LIN {X 0,Y 452.591,Z 786.867,A -85,B 0,C 180,E1 7857.223,E2 7857.223} C_VEL
LIN {X 0,Y 442.447,Z 754.81,A -85,B 0,C 180,E1 7858.353,E2 7858.353} C_VEL
LIN {X 0,Y 442.001,Z 754.81,A -85,B 0,C 180,E1 7869.434,E2 7869.434} C_VEL
LIN {X 0,Y 441.88,Z 754.81,A -85,B 0,C 180,E1 7877.96,E2 7877.96} C_VEL
LIN {X 0,Y 441.928,Z 754.81,A -85,B 0,C 180,E1 7887.845,E2 7887.845} C_VEL
LIN {X 0,Y 442.308,Z 754.81,A -85,B 0,C 180,E1 7898.887,E2 7898.887} C_VEL
LIN {X 0,Y 442.704,Z 754.81,A -85,B 0,C 180,E1 7909.135,E2 7909.135} C_VEL
LIN {X 0,Y 443.031,Z 754.81,A -85,B 0,C 180,E1 7919.021,E2 7919.021} C_VEL
LIN {X 0,Y 442.966,Z 754.81,A -85,B 0,C 180,E1 7928.871,E2 7928.871} C_VEL
LIN {X 0,Y 442.439,Z 754.81,A -85,B 0,C 180,E1 7939.392,E2 7939.392} C_VEL
LIN {X 0,Y 442.078,Z 754.81,A -85,B 0,C 180,E1 7949.854,E2 7949.854} C_VEL
LIN {X 0,Y 441.847,Z 754.81,A -85,B 0,C 180,E1 7959.452,E2 7959.452} C_VEL
LIN {X 0,Y 441.828,Z 754.81,A -85,B 0,C 180,E1 7967.949,E2 7967.949} C_VEL
LIN {X 0,Y 441.919,Z 754.81,A -85,B 0,C 180,E1 7977.84,E2 7977.84} C_VEL
LIN {X 0,Y 441.903,Z 754.81,A -85,B 0,C 180,E1 7986.738,E2 7986.738} C_VEL
LIN {X 0,Y 442.395,Z 754.81,A -85,B 0,C 180,E1 7997.116,E2 7997.116} C_VEL
LIN {X 0,Y 443.108,Z 754.81,A -85,B 0,C 180,E1 8007.055,E2 8007.055} C_VEL
LIN {X 0,Y 442.368,Z 756.655,A -85,B 0,C 180,E1 8012.365,E2 8012.365} C_VEL
LIN {X 0,Y 449.575,Z 792.358,A -85,B 0,C 180,E1 8014.536,E2 8014.536} C_VEL
LIN {X 0,Y 447.004,Z 827.238,A -85,B 0,C 180,E1 8018.05,E2 8018.05} C_VEL
LIN {X 0,Y 445.134,Z 851.284,A -85,B 0,C 180,E1 8022.802,E2 8022.802} C_VEL
LIN {X 0,Y 444.477,Z 860.925,A -85,B 0,C 180,E1 8026.87,E2 8026.87} C_VEL
LIN {X 0,Y 444.267,Z 862.934,A -85,B 0,C 180,E1 8031.018,E2 8031.018} C_VEL
LIN {X 0,Y 445.039,Z 852.888,A -85,B 0,C 180,E1 8036.859,E2 8036.859} C_VEL
LIN {X 0,Y 447.157,Z 829.66,A -85,B 0,C 180,E1 8041.738,E2 8041.738} C_VEL
LIN {X 0,Y 449.893,Z 795.07,A -85,B 0,C 180,E1 8045.397,E2 8045.397} C_VEL
LIN {X 0,Y 445.984,Z 767.35,A -85,B 0,C 180,E1 8047.255,E2 8047.255} C_VEL
LIN {X 0,Y 442.165,Z 754.81,A -85,B 0,C 180,E1 8048.173,E2 8048.173} C_VEL
LIN {X 0,Y 441.871,Z 754.81,A -85,B 0,C 180,E1 8057.953,E2 8057.953} C_VEL
LIN {X 0,Y 441.961,Z 754.81,A -85,B 0,C 180,E1 8067.842,E2 8067.842} C_VEL
LIN {X 0,Y 441.936,Z 754.81,A -85,B 0,C 180,E1 8076.738,E2 8076.738} C_VEL
LIN {X 0,Y 442.368,Z 754.81,A -85,B 0,C 180,E1 8087.113,E2 8087.113} C_VEL
LIN {X 0,Y 443.223,Z 754.81,A -85,B 0,C 180,E1 8097.919,E2 8097.919} C_VEL
LIN {X 0,Y 442.747,Z 754.81,A -85,B 0,C 180,E1 8108.87,E2 8108.87} C_VEL
LIN {X 0,Y 442.392,Z 754.81,A -85,B 0,C 180,E1 8119.379,E2 8119.379} C_VEL
LIN {X 0,Y 442.145,Z 754.81,A -85,B 0,C 180,E1 8129.843,E2 8129.843} C_VEL
LIN {X 0,Y 442.036,Z 754.81,A -85,B 0,C 180,E1 8139.426,E2 8139.426} C_VEL
LIN {X 0,Y 441.905,Z 754.81,A -85,B 0,C 180,E1 8147.96,E2 8147.96} C_VEL
LIN {X 0,Y 441.987,Z 754.81,A -85,B 0,C 180,E1 8157.847,E2 8157.847} C_VEL
LIN {X 0,Y 442.617,Z 756.744,A -85,B 0,C 180,E1 8161.684,E2 8161.684} C_VEL
LIN {X 0,Y 454.951,Z 801.269,A -85,B 0,C 180,E1 8163.103,E2 8163.103} C_VEL
LIN {X 0,Y 452.795,Z 857.855,A -85,B 0,C 180,E1 8164.779,E2 8164.779} C_VEL
LIN {X 0,Y 442.938,Z 889.427,A -85,B 0,C 180,E1 8166.427,E2 8166.427} C_VEL
LIN {X 0,Y 438.726,Z 935.255,A -85,B 0,C 180,E1 8171.199,E2 8171.199} C_VEL
LIN {X 0,Y 436.456,Z 968.703,A -85,B 0,C 180,E1 8177.194,E2 8177.194} C_VEL
LIN {X 0,Y 436.059,Z 988.848,A -85,B 0,C 180,E1 8184.008,E2 8184.008} C_VEL
LIN {X 0,Y 435.858,Z 994.128,A -85,B 0,C 180,E1 8190.998,E2 8190.998} C_VEL
LIN {X 0,Y 435.692,Z 985.83,A -85,B 0,C 180,E1 8197.506,E2 8197.506} C_VEL
LIN {X 0,Y 436.647,Z 963.898,A -85,B 0,C 180,E1 8203.956,E2 8203.956} C_VEL
LIN {X 0,Y 439.499,Z 927.872,A -85,B 0,C 180,E1 8209.806,E2 8209.806} C_VEL
LIN {X 0,Y 443.485,Z 882.164,A -85,B 0,C 180,E1 8214.111,E2 8214.111} C_VEL
LIN {X 0,Y 446.96,Z 829.737,A -85,B 0,C 180,E1 8216.636,E2 8216.636} C_VEL
LIN {X 0,Y 445.096,Z 788.288,A -85,B 0,C 180,E1 8217.571,E2 8217.571} C_VEL
LIN {X 0,Y 434.362,Z 754.81,A -85,B 0,C 180,E1 8218.782,E2 8218.782} C_VEL
LIN {X 0,Y 433.933,Z 754.81,A -85,B 0,C 180,E1 8228.11,E2 8228.11} C_VEL
LIN {X 0,Y 433.819,Z 754.81,A -85,B 0,C 180,E1 8238.774,E2 8238.774} C_VEL
LIN {X 0,Y 433.954,Z 754.81,A -85,B 0,C 180,E1 8249.534,E2 8249.534} C_VEL
LIN {X 0,Y 434.39,Z 754.81,A -85,B 0,C 180,E1 8260.62,E2 8260.62} C_VEL
LIN {X 0,Y 434.769,Z 754.81,A -85,B 0,C 180,E1 8270.966,E2 8270.966} C_VEL
LIN {X 0,Y 435.526,Z 754.81,A -85,B 0,C 180,E1 8281.001,E2 8281.001} C_VEL
LIN {X 0,Y 434.752,Z 754.81,A -85,B 0,C 180,E1 8291.071,E2 8291.071} C_VEL
LIN {X 0,Y 434.339,Z 754.81,A -85,B 0,C 180,E1 8301.525,E2 8301.525} C_VEL
LIN {X 0,Y 433.906,Z 754.81,A -85,B 0,C 180,E1 8311.031,E2 8311.031} C_VEL
LIN {X 0,Y 433.754,Z 754.81,A -85,B 0,C 180,E1 8321.216,E2 8321.216} C_VEL
LIN {X 0,Y 433.694,Z 754.81,A -85,B 0,C 180,E1 8331.938,E2 8331.938} C_VEL
LIN {X 0,Y 433.989,Z 754.81,A -85,B 0,C 180,E1 8341.831,E2 8341.831} C_VEL
LIN {X 0,Y 434.256,Z 754.81,A -85,B 0,C 180,E1 8352.719,E2 8352.719} C_VEL
LIN {X 0,Y 434.917,Z 754.81,A -85,B 0,C 180,E1 8362.984,E2 8362.984} C_VEL
LIN {X 0,Y 434.264,Z 754.81,A -85,B 0,C 180,E1 8371.877,E2 8371.877} C_VEL
LIN {X 0,Y 441.972,Z 793.979,A -85,B 0,C 180,E1 8374.278,E2 8374.278} C_VEL
LIN {X 0,Y 439.206,Z 829.188,A -85,B 0,C 180,E1 8377.944,E2 8377.944} C_VEL
LIN {X 0,Y 437.188,Z 853.627,A -85,B 0,C 180,E1 8383.039,E2 8383.039} C_VEL
LIN {X 0,Y 436.52,Z 862.544,A -85,B 0,C 180,E1 8387.187,E2 8387.187} C_VEL
LIN {X 0,Y 436.714,Z 861.813,A -85,B 0,C 180,E1 8393.554,E2 8393.554} C_VEL
LIN {X 0,Y 438.444,Z 845.603,A -85,B 0,C 180,E1 8399.268,E2 8399.268} C_VEL
LIN {X 0,Y 441.034,Z 816.527,A -85,B 0,C 180,E1 8403.848,E2 8403.848} C_VEL
LIN {X 0,Y 441.317,Z 779.381,A -85,B 0,C 180,E1 8406.941,E2 8406.941} C_VEL
LIN {X 0,Y 434.105,Z 754.81,A -85,B 0,C 180,E1 8408.698,E2 8408.698} C_VEL
LIN {X 0,Y 433.757,Z 754.81,A -85,B 0,C 180,E1 8419.663,E2 8419.663} C_VEL
LIN {X 0,Y 433.983,Z 754.81,A -85,B 0,C 180,E1 8429.531,E2 8429.531} C_VEL
LIN {X 0,Y 434.05,Z 754.81,A -85,B 0,C 180,E1 8440.598,E2 8440.598} C_VEL
LIN {X 0,Y 434.799,Z 754.81,A -85,B 0,C 180,E1 8450.961,E2 8450.961} C_VEL
LIN {X 0,Y 435.015,Z 754.81,A -85,B 0,C 180,E1 8460.997,E2 8460.997} C_VEL
LIN {X 0,Y 434.668,Z 754.81,A -85,B 0,C 180,E1 8471.068,E2 8471.068} C_VEL
LIN {X 0,Y 434.322,Z 754.81,A -85,B 0,C 180,E1 8481.52,E2 8481.52} C_VEL
LIN {X 0,Y 433.999,Z 754.81,A -85,B 0,C 180,E1 8491.054,E2 8491.054} C_VEL
LIN {X 0,Y 433.921,Z 754.81,A -85,B 0,C 180,E1 8501.243,E2 8501.243} C_VEL
LIN {X 0,Y 433.89,Z 754.81,A -85,B 0,C 180,E1 8512.261,E2 8512.261} C_VEL
LIN {X 0,Y 434.389,Z 756.03,A -85,B 0,C 180,E1 8521.168,E2 8521.168} C_VEL
LIN {X 0,Y 447.578,Z 800.376,A -85,B 0,C 180,E1 8522.692,E2 8522.692} C_VEL
LIN {X 0,Y 445.33,Z 857.166,A -85,B 0,C 180,E1 8524.398,E2 8524.398} C_VEL
LIN {X 0,Y 442.938,Z 889.427,A -85,B 0,C 180,E1 8526.427,E2 8526.427} C_VEL
LIN {X 0,Y 432.598,Z 917.951,A -85,B 0,C 180,E1 8528.842,E2 8528.842} C_VEL
LIN {X 0,Y 429.325,Z 956.761,A -85,B 0,C 180,E1 8534.627,E2 8534.627} C_VEL
LIN {X 0,Y 427.9,Z 982.008,A -85,B 0,C 180,E1 8541.331,E2 8541.331} C_VEL
LIN {X 0,Y 427.815,Z 991.674,A -85,B 0,C 180,E1 8546.951,E2 8546.951} C_VEL
LIN {X 0,Y 428.118,Z 990.75,A -85,B 0,C 180,E1 8554.066,E2 8554.066} C_VEL
LIN {X 0,Y 428.165,Z 974.434,A -85,B 0,C 180,E1 8561.242,E2 8561.242} C_VEL
LIN {X 0,Y 430.13,Z 944.424,A -85,B 0,C 180,E1 8567.613,E2 8567.613} C_VEL
LIN {X 0,Y 434.112,Z 902.67,A -85,B 0,C 180,E1 8572.723,E2 8572.723} C_VEL
LIN {X 0,Y 438.158,Z 851.791,A -85,B 0,C 180,E1 8576.165,E2 8576.165} C_VEL
LIN {X 0,Y 439.043,Z 794.483,A -85,B 0,C 180,E1 8577.778,E2 8577.778} C_VEL
LIN {X 0,Y 426.256,Z 754.81,A -85,B 0,C 180,E1 8579.285,E2 8579.285} C_VEL
LIN {X 0,Y 425.858,Z 754.81,A -85,B 0,C 180,E1 8589.994,E2 8589.994} C_VEL
LIN {X 0,Y 425.782,Z 754.81,A -85,B 0,C 180,E1 8600.024,E2 8600.024} C_VEL
LIN {X 0,Y 425.936,Z 754.81,A -85,B 0,C 180,E1 8611.253,E2 8611.253} C_VEL
LIN {X 0,Y 426.384,Z 754.81,A -85,B 0,C 180,E1 8622.393,E2 8622.393} C_VEL
LIN {X 0,Y 426.997,Z 754.81,A -85,B 0,C 180,E1 8632.857,E2 8632.857} C_VEL
LIN {X 0,Y 427.048,Z 754.81,A -85,B 0,C 180,E1 8643.058,E2 8643.058} C_VEL
LIN {X 0,Y 426.644,Z 754.81,A -85,B 0,C 180,E1 8653.37,E2 8653.37} C_VEL
LIN {X 0,Y 426.194,Z 754.81,A -85,B 0,C 180,E1 8664.175,E2 8664.175} C_VEL
LIN {X 0,Y 425.794,Z 754.81,A -85,B 0,C 180,E1 8673.537,E2 8673.537} C_VEL
LIN {X 0,Y 425.737,Z 754.81,A -85,B 0,C 180,E1 8684.037,E2 8684.037} C_VEL
LIN {X 0,Y 425.708,Z 754.81,A -85,B 0,C 180,E1 8693.97,E2 8693.97} C_VEL
LIN {X 0,Y 425.968,Z 754.81,A -85,B 0,C 180,E1 8703.555,E2 8703.555} C_VEL
LIN {X 0,Y 426.32,Z 754.81,A -85,B 0,C 180,E1 8714.515,E2 8714.515} C_VEL
LIN {X 0,Y 426.825,Z 754.81,A -85,B 0,C 180,E1 8724.9,E2 8724.9} C_VEL
LIN {X 0,Y 426.509,Z 756.493,A -85,B 0,C 180,E1 8731.529,E2 8731.529} C_VEL
LIN {X 0,Y 434.337,Z 795.975,A -85,B 0,C 180,E1 8734.038,E2 8734.038} C_VEL
LIN {X 0,Y 431.444,Z 831.116,A -85,B 0,C 180,E1 8737.833,E2 8737.833} C_VEL
LIN {X 0,Y 429.385,Z 854.31,A -85,B 0,C 180,E1 8742.761,E2 8742.761} C_VEL
LIN {X 0,Y 428.56,Z 864.155,A -85,B 0,C 180,E1 8747.517,E2 8747.517} C_VEL
LIN {X 0,Y 428.808,Z 863.488,A -85,B 0,C 180,E1 8753.308,E2 8753.308} C_VEL
LIN {X 0,Y 430.356,Z 849.139,A -85,B 0,C 180,E1 8758.923,E2 8758.923} C_VEL
LIN {X 0,Y 433.012,Z 822.26,A -85,B 0,C 180,E1 8763.619,E2 8763.619} C_VEL
LIN {X 0,Y 434.797,Z 785.115,A -85,B 0,C 180,E1 8767.001,E2 8767.001} C_VEL
LIN {X 0,Y 426.077,Z 754.81,A -85,B 0,C 180,E1 8769.059,E2 8769.059} C_VEL
LIN {X 0,Y 425.729,Z 754.81,A -85,B 0,C 180,E1 8780.031,E2 8780.031} C_VEL
LIN {X 0,Y 425.972,Z 754.81,A -85,B 0,C 180,E1 8791.25,E2 8791.25} C_VEL
LIN {X 0,Y 426.174,Z 754.81,A -85,B 0,C 180,E1 8802.379,E2 8802.379} C_VEL
LIN {X 0,Y 426.87,Z 754.81,A -85,B 0,C 180,E1 8812.85,E2 8812.85} C_VEL
LIN {X 0,Y 427.024,Z 754.81,A -85,B 0,C 180,E1 8821.016,E2 8821.016} C_VEL
LIN {X 0,Y 426.647,Z 754.81,A -85,B 0,C 180,E1 8831.279,E2 8831.279} C_VEL
LIN {X 0,Y 426.291,Z 754.81,A -85,B 0,C 180,E1 8841.947,E2 8841.947} C_VEL
LIN {X 0,Y 425.989,Z 754.81,A -85,B 0,C 180,E1 8853.157,E2 8853.157} C_VEL
LIN {X 0,Y 425.864,Z 754.81,A -85,B 0,C 180,E1 8864.014,E2 8864.014} C_VEL
LIN {X 0,Y 425.834,Z 754.81,A -85,B 0,C 180,E1 8873.984,E2 8873.984} C_VEL
LIN {X 0,Y 426.437,Z 756.637,A -85,B 0,C 180,E1 8880.672,E2 8880.672} C_VEL
LIN {X 0,Y 440.238,Z 802.364,A -85,B 0,C 180,E1 8882.317,E2 8882.317} C_VEL
LIN {X 0,Y 437.767,Z 857.949,A -85,B 0,C 180,E1 8884.077,E2 8884.077} C_VEL
LIN {X 0,Y 433.688,Z 907.236,A -85,B 0,C 180,E1 8887.711,E2 8887.711} C_VEL
LIN {X 0,Y 432.598,Z 917.951,A -85,B 0,C 180,E1 8888.842,E2 8888.842} C_VEL
LIN {X 0,Y 422.426,Z 942.481,A -85,B 0,C 180,E1 8891.991,E2 8891.991} C_VEL
LIN {X 0,Y 420.454,Z 973.012,A -85,B 0,C 180,E1 8898.551,E2 8898.551} C_VEL
LIN {X 0,Y 420.028,Z 989.458,A -85,B 0,C 180,E1 8905.857,E2 8905.857} C_VEL
LIN {X 0,Y 420.02,Z 991.768,A -85,B 0,C 180,E1 8911.036,E2 8911.036} C_VEL
LIN {X 0,Y 419.857,Z 983.376,A -85,B 0,C 180,E1 8917.791,E2 8917.791} C_VEL
LIN {X 0,Y 421.142,Z 959.449,A -85,B 0,C 180,E1 8924.878,E2 8924.878} C_VEL
LIN {X 0,Y 424.355,Z 922.522,A -85,B 0,C 180,E1 8930.818,E2 8930.818} C_VEL
LIN {X 0,Y 428.776,Z 874.925,A -85,B 0,C 180,E1 8935.196,E2 8935.196} C_VEL
LIN {X 0,Y 432.221,Z 822.667,A -85,B 0,C 180,E1 8937.566,E2 8937.566} C_VEL
LIN {X 0,Y 430.033,Z 790.74,A -85,B 0,C 180,E1 8938.316,E2 8938.316} C_VEL
LIN {X 0,Y 418.191,Z 754.81,A -85,B 0,C 180,E1 8939.739,E2 8939.739} C_VEL
LIN {X 0,Y 417.841,Z 754.81,A -85,B 0,C 180,E1 8949.465,E2 8949.465} C_VEL
LIN {X 0,Y 417.763,Z 754.81,A -85,B 0,C 180,E1 8960.532,E2 8960.532} C_VEL
LIN {X 0,Y 417.91,Z 754.81,A -85,B 0,C 180,E1 8970.648,E2 8970.648} C_VEL
LIN {X 0,Y 418.354,Z 754.81,A -85,B 0,C 180,E1 8982.044,E2 8982.044} C_VEL
LIN {X 0,Y 418.979,Z 754.81,A -85,B 0,C 180,E1 8992.72,E2 8992.72} C_VEL
LIN {X 0,Y 419.031,Z 754.81,A -85,B 0,C 180,E1 9003.117,E2 9003.117} C_VEL
LIN {X 0,Y 418.611,Z 754.81,A -85,B 0,C 180,E1 9013.632,E2 9013.632} C_VEL
LIN {X 0,Y 418.182,Z 754.81,A -85,B 0,C 180,E1 9024.669,E2 9024.669} C_VEL
LIN {X 0,Y 417.626,Z 754.81,A -85,B 0,C 180,E1 9035.153,E2 9035.153} C_VEL
LIN {X 0,Y 417.7,Z 754.81,A -85,B 0,C 180,E1 9045.113,E2 9045.113} C_VEL
LIN {X 0,Y 417.703,Z 754.81,A -85,B 0,C 180,E1 9055.726,E2 9055.726} C_VEL
LIN {X 0,Y 417.905,Z 754.81,A -85,B 0,C 180,E1 9065.316,E2 9065.316} C_VEL
LIN {X 0,Y 418.308,Z 754.81,A -85,B 0,C 180,E1 9076.36,E2 9076.36} C_VEL
LIN {X 0,Y 419.055,Z 754.81,A -85,B 0,C 180,E1 9086.885,E2 9086.885} C_VEL
LIN {X 0,Y 418.638,Z 756.628,A -85,B 0,C 180,E1 9091.103,E2 9091.103} C_VEL
LIN {X 0,Y 426.819,Z 796.423,A -85,B 0,C 180,E1 9093.676,E2 9093.676} C_VEL
LIN {X 0,Y 423.789,Z 831.313,A -85,B 0,C 180,E1 9097.458,E2 9097.458} C_VEL
LIN {X 0,Y 421.581,Z 854.962,A -85,B 0,C 180,E1 9102.473,E2 9102.473} C_VEL
LIN {X 0,Y 420.616,Z 865.658,A -85,B 0,C 180,E1 9107.858,E2 9107.858} C_VEL
LIN {X 0,Y 421.087,Z 863.073,A -85,B 0,C 180,E1 9114.484,E2 9114.484} C_VEL
LIN {X 0,Y 423.127,Z 846.139,A -85,B 0,C 180,E1 9120.133,E2 9120.133} C_VEL
LIN {X 0,Y 426.134,Z 817.816,A -85,B 0,C 180,E1 9124.615,E2 9124.615} C_VEL
LIN {X 0,Y 426.482,Z 782.61,A -85,B 0,C 180,E1 9127.696,E2 9127.696} C_VEL
LIN {X 0,Y 417.977,Z 754.81,A -85,B 0,C 180,E1 9129.796,E2 9129.796} C_VEL
LIN {X 0,Y 417.703,Z 754.81,A -85,B 0,C 180,E1 9140.518,E2 9140.518} C_VEL
LIN {X 0,Y 417.943,Z 754.81,A -85,B 0,C 180,E1 9150.644,E2 9150.644} C_VEL
LIN {X 0,Y 418.123,Z 754.81,A -85,B 0,C 180,E1 9162.028,E2 9162.028} C_VEL
LIN {X 0,Y 418.851,Z 754.81,A -85,B 0,C 180,E1 9172.712,E2 9172.712} C_VEL
LIN {X 0,Y 419.017,Z 754.81,A -85,B 0,C 180,E1 9181.035,E2 9181.035} C_VEL
LIN {X 0,Y 418.648,Z 754.81,A -85,B 0,C 180,E1 9191.497,E2 9191.497} C_VEL
LIN {X 0,Y 418.226,Z 754.81,A -85,B 0,C 180,E1 9202.393,E2 9202.393} C_VEL
LIN {X 0,Y 417.933,Z 754.81,A -85,B 0,C 180,E1 9211.767,E2 9211.767} C_VEL
LIN {X 0,Y 417.864,Z 754.81,A -85,B 0,C 180,E1 9222.207,E2 9222.207} C_VEL
LIN {X 0,Y 417.835,Z 754.81,A -85,B 0,C 180,E1 9233.183,E2 9233.183} C_VEL
LIN {X 0,Y 418.284,Z 756.272,A -85,B 0,C 180,E1 9240.119,E2 9240.119} C_VEL
LIN {X 0,Y 432.955,Z 804.082,A -85,B 0,C 180,E1 9241.912,E2 9241.912} C_VEL
LIN {X 0,Y 430.197,Z 858.79,A -85,B 0,C 180,E1 9243.743,E2 9243.743} C_VEL
LIN {X 0,Y 425.718,Z 908.98,A -85,B 0,C 180,E1 9247.615,E2 9247.615} C_VEL
LIN {X 0,Y 422.426,Z 942.481,A -85,B 0,C 180,E1 9251.991,E2 9251.991} C_VEL
LIN {X 0,Y 412.724,Z 962.347,A -85,B 0,C 180,E1 9255.822,E2 9255.822} C_VEL
LIN {X 0,Y 412.01,Z 983.167,A -85,B 0,C 180,E1 9262.594,E2 9262.594} C_VEL
LIN {X 0,Y 412.291,Z 990.591,A -85,B 0,C 180,E1 9268.946,E2 9268.946} C_VEL
LIN {X 0,Y 412.076,Z 986.99,A -85,B 0,C 180,E1 9275.283,E2 9275.283} C_VEL
LIN {X 0,Y 412.259,Z 969.907,A -85,B 0,C 180,E1 9282.239,E2 9282.239} C_VEL
LIN {X 0,Y 414.602,Z 938.989,A -85,B 0,C 180,E1 9288.68,E2 9288.68} C_VEL
LIN {X 0,Y 419.144,Z 895.529,A -85,B 0,C 180,E1 9293.896,E2 9293.896} C_VEL
LIN {X 0,Y 423.48,Z 845.445,A -85,B 0,C 180,E1 9297.149,E2 9297.149} C_VEL
LIN {X 0,Y 423.087,Z 794.106,A -85,B 0,C 180,E1 9298.626,E2 9298.626} C_VEL
LIN {X 0,Y 410.116,Z 754.81,A -85,B 0,C 180,E1 9300.236,E2 9300.236} C_VEL
LIN {X 0,Y 409.752,Z 754.81,A -85,B 0,C 180,E1 9310.608,E2 9310.608} C_VEL
LIN {X 0,Y 409.693,Z 754.81,A -85,B 0,C 180,E1 9319.596,E2 9319.596} C_VEL
LIN {X 0,Y 409.889,Z 754.81,A -85,B 0,C 180,E1 9330.468,E2 9330.468} C_VEL
LIN {X 0,Y 410.292,Z 754.81,A -85,B 0,C 180,E1 9341.679,E2 9341.679} C_VEL
LIN {X 0,Y 410.939,Z 754.81,A -85,B 0,C 180,E1 9352.576,E2 9352.576} C_VEL
LIN {X 0,Y 411.028,Z 754.81,A -85,B 0,C 180,E1 9363.177,E2 9363.177} C_VEL
LIN {X 0,Y 410.573,Z 754.81,A -85,B 0,C 180,E1 9373.904,E2 9373.904} C_VEL
LIN {X 0,Y 410.104,Z 754.81,A -85,B 0,C 180,E1 9385.188,E2 9385.188} C_VEL
LIN {X 0,Y 409.635,Z 754.81,A -85,B 0,C 180,E1 9395.048,E2 9395.048} C_VEL
LIN {X 0,Y 409.604,Z 754.81,A -85,B 0,C 180,E1 9406.262,E2 9406.262} C_VEL
LIN {X 0,Y 409.714,Z 754.81,A -85,B 0,C 180,E1 9417.514,E2 9417.514} C_VEL
LIN {X 0,Y 409.823,Z 754.81,A -85,B 0,C 180,E1 9427.118,E2 9427.118} C_VEL
LIN {X 0,Y 410.474,Z 754.81,A -85,B 0,C 180,E1 9438.455,E2 9438.455} C_VEL
LIN {X 0,Y 411.317,Z 754.81,A -85,B 0,C 180,E1 9448.942,E2 9448.942} C_VEL
LIN {X 0,Y 410.806,Z 756.741,A -85,B 0,C 180,E1 9450.661,E2 9450.661} C_VEL
LIN {X 0,Y 419.227,Z 798.212,A -85,B 0,C 180,E1 9453.413,E2 9453.413} C_VEL
LIN {X 0,Y 415.998,Z 833.178,A -85,B 0,C 180,E1 9457.335,E2 9457.335} C_VEL
LIN {X 0,Y 413.678,Z 856.697,A -85,B 0,C 180,E1 9462.529,E2 9462.529} C_VEL
LIN {X 0,Y 412.673,Z 867.156,A -85,B 0,C 180,E1 9468.214,E2 9468.214} C_VEL
LIN {X 0,Y 413.309,Z 863.652,A -85,B 0,C 180,E1 9474.976,E2 9474.976} C_VEL
LIN {X 0,Y 415.625,Z 845.043,A -85,B 0,C 180,E1 9480.897,E2 9480.897} C_VEL
LIN {X 0,Y 419.094,Z 814.777,A -85,B 0,C 180,E1 9485.435,E2 9485.435} C_VEL
LIN {X 0,Y 419.03,Z 784.069,A -85,B 0,C 180,E1 9488.107,E2 9488.107} C_VEL
LIN {X 0,Y 409.923,Z 754.81,A -85,B 0,C 180,E1 9490.38,E2 9490.38} C_VEL
LIN {X 0,Y 409.652,Z 754.81,A -85,B 0,C 180,E1 9499.584,E2 9499.584} C_VEL
LIN {X 0,Y 409.933,Z 754.81,A -85,B 0,C 180,E1 9510.454,E2 9510.454} C_VEL
LIN {X 0,Y 410.046,Z 754.81,A -85,B 0,C 180,E1 9521.662,E2 9521.662} C_VEL
LIN {X 0,Y 410.821,Z 754.81,A -85,B 0,C 180,E1 9532.569,E2 9532.569} C_VEL
LIN {X 0,Y 411.027,Z 754.81,A -85,B 0,C 180,E1 9541.055,E2 9541.055} C_VEL
LIN {X 0,Y 410.63,Z 754.81,A -85,B 0,C 180,E1 9551.725,E2 9551.725} C_VEL
LIN {X 0,Y 410.162,Z 754.81,A -85,B 0,C 180,E1 9562.857,E2 9562.857} C_VEL
LIN {X 0,Y 409.842,Z 754.81,A -85,B 0,C 180,E1 9573.579,E2 9573.579} C_VEL
LIN {X 0,Y 409.716,Z 754.81,A -85,B 0,C 180,E1 9583.758,E2 9583.758} C_VEL
LIN {X 0,Y 409.813,Z 754.81,A -85,B 0,C 180,E1 9594.973,E2 9594.973} C_VEL
LIN {X 0,Y 410.193,Z 756.226,A -85,B 0,C 180,E1 9599.538,E2 9599.538} C_VEL
LIN {X 0,Y 425.692,Z 805.295,A -85,B 0,C 180,E1 9601.484,E2 9601.484} C_VEL
LIN {X 0,Y 422.661,Z 859.766,A -85,B 0,C 180,E1 9603.4,E2 9603.4} C_VEL
LIN {X 0,Y 418.017,Z 908.692,A -85,B 0,C 180,E1 9607.312,E2 9607.312} C_VEL
LIN {X 0,Y 414.12,Z 948.974,A -85,B 0,C 180,E1 9613.013,E2 9613.013} C_VEL
LIN {X 0,Y 412.724,Z 962.347,A -85,B 0,C 180,E1 9615.822,E2 9615.822} C_VEL
LIN {X 0,Y 404.251,Z 976.838,A -85,B 0,C 180,E1 9620.231,E2 9620.231} C_VEL
LIN {X 0,Y 404.086,Z 988.13,A -85,B 0,C 180,E1 9626.771,E2 9626.771} C_VEL
LIN {X 0,Y 404.216,Z 988.182,A -85,B 0,C 180,E1 9633.229,E2 9633.229} C_VEL
LIN {X 0,Y 404.288,Z 973.923,A -85,B 0,C 180,E1 9640.818,E2 9640.818} C_VEL
LIN {X 0,Y 406.174,Z 945.392,A -85,B 0,C 180,E1 9647.696,E2 9647.696} C_VEL
LIN {X 0,Y 410.528,Z 904.705,A -85,B 0,C 180,E1 9653.272,E2 9653.272} C_VEL
LIN {X 0,Y 415.161,Z 855.742,A -85,B 0,C 180,E1 9657.009,E2 9657.009} C_VEL
LIN {X 0,Y 417.289,Z 800.971,A -85,B 0,C 180,E1 9658.822,E2 9658.822} C_VEL
LIN {X 0,Y 402.086,Z 754.81,A -85,B 0,C 180,E1 9660.633,E2 9660.633} C_VEL
LIN {X 0,Y 401.652,Z 754.81,A -85,B 0,C 180,E1 9671.393,E2 9671.393} C_VEL
LIN {X 0,Y 401.636,Z 754.81,A -85,B 0,C 180,E1 9681.436,E2 9681.436} C_VEL
LIN {X 0,Y 401.899,Z 754.81,A -85,B 0,C 180,E1 9692.545,E2 9692.545} C_VEL
LIN {X 0,Y 402.435,Z 754.81,A -85,B 0,C 180,E1 9704.073,E2 9704.073} C_VEL
LIN {X 0,Y 403,Z 754.81,A -85,B 0,C 180,E1 9714.601,E2 9714.601} C_VEL
LIN {X 0,Y 402.965,Z 754.81,A -85,B 0,C 180,E1 9723.618,E2 9723.618} C_VEL
LIN {X 0,Y 402.537,Z 754.81,A -85,B 0,C 180,E1 9734.187,E2 9734.187} C_VEL
LIN {X 0,Y 402.008,Z 754.81,A -85,B 0,C 180,E1 9745.732,E2 9745.732} C_VEL
LIN {X 0,Y 401.594,Z 754.81,A -85,B 0,C 180,E1 9755.857,E2 9755.857} C_VEL
LIN {X 0,Y 401.541,Z 754.81,A -85,B 0,C 180,E1 9765.637,E2 9765.637} C_VEL
LIN {X 0,Y 401.68,Z 754.81,A -85,B 0,C 180,E1 9776.782,E2 9776.782} C_VEL
LIN {X 0,Y 401.776,Z 754.81,A -85,B 0,C 180,E1 9787.734,E2 9787.734} C_VEL
LIN {X 0,Y 402.372,Z 754.81,A -85,B 0,C 180,E1 9798.027,E2 9798.027} C_VEL
LIN {X 0,Y 403.308,Z 754.81,A -85,B 0,C 180,E1 9808.921,E2 9808.921} C_VEL
LIN {X 0,Y 402.997,Z 756.719,A -85,B 0,C 180,E1 9810.202,E2 9810.202} C_VEL
LIN {X 0,Y 411.711,Z 798.72,A -85,B 0,C 180,E1 9813.038,E2 9813.038} C_VEL
LIN {X 0,Y 408.204,Z 834.99,A -85,B 0,C 180,E1 9817.207,E2 9817.207} C_VEL
LIN {X 0,Y 405.732,Z 858.628,A -85,B 0,C 180,E1 9822.671,E2 9822.671} C_VEL
LIN {X 0,Y 404.754,Z 868.556,A -85,B 0,C 180,E1 9828.583,E2 9828.583} C_VEL
LIN {X 0,Y 405.499,Z 864.194,A -85,B 0,C 180,E1 9835.491,E2 9835.491} C_VEL
LIN {X 0,Y 408.027,Z 845.328,A -85,B 0,C 180,E1 9841.364,E2 9841.364} C_VEL
LIN {X 0,Y 411.791,Z 814.569,A -85,B 0,C 180,E1 9845.958,E2 9845.958} C_VEL
LIN {X 0,Y 411.439,Z 784.862,A -85,B 0,C 180,E1 9848.6,E2 9848.6} C_VEL
LIN {X 0,Y 401.862,Z 754.81,A -85,B 0,C 180,E1 9850.93,E2 9850.93} C_VEL
LIN {X 0,Y 401.554,Z 754.81,A -85,B 0,C 180,E1 9861.419,E2 9861.419} C_VEL
LIN {X 0,Y 401.921,Z 754.81,A -85,B 0,C 180,E1 9872.536,E2 9872.536} C_VEL
LIN {X 0,Y 402.205,Z 754.81,A -85,B 0,C 180,E1 9884.183,E2 9884.183} C_VEL
LIN {X 0,Y 402.777,Z 754.81,A -85,B 0,C 180,E1 9894.592,E2 9894.592} C_VEL
LIN {X 0,Y 402.859,Z 754.81,A -85,B 0,C 180,E1 9903.395,E2 9903.395} C_VEL
LIN {X 0,Y 402.511,Z 754.81,A -85,B 0,C 180,E1 9914.183,E2 9914.183} C_VEL
LIN {X 0,Y 402.019,Z 754.81,A -85,B 0,C 180,E1 9925.725,E2 9925.725} C_VEL
LIN {X 0,Y 401.854,Z 754.81,A -85,B 0,C 180,E1 9935.823,E2 9935.823} C_VEL
LIN {X 0,Y 401.625,Z 754.81,A -85,B 0,C 180,E1 9947.456,E2 9947.456} C_VEL
LIN {X 0,Y 402.141,Z 756.322,A -85,B 0,C 180,E1 9958.936,E2 9958.936} C_VEL
LIN {X 0,Y 418.44,Z 806.325,A -85,B 0,C 180,E1 9961.041,E2 9961.041} C_VEL
LIN {X 0,Y 415.096,Z 860.998,A -85,B 0,C 180,E1 9963.069,E2 9963.069} C_VEL
LIN {X 0,Y 410.139,Z 909.749,A -85,B 0,C 180,E1 9967.139,E2 9967.139} C_VEL
LIN {X 0,Y 406.149,Z 949.193,A -85,B 0,C 180,E1 9972.97,E2 9972.97} C_VEL
LIN {X 0,Y 404.251,Z 976.838,A -85,B 0,C 180,E1 9980.231,E2 9980.231} C_VEL
LIN {X 0,Y 396.308,Z 985.239,A -85,B 0,C 180,E1 9985.053,E2 9985.053} C_VEL
LIN {X 0,Y 396.278,Z 988.222,A -85,B 0,C 180,E1 9991.098,E2 9991.098} C_VEL
LIN {X 0,Y 396.126,Z 979.622,A -85,B 0,C 180,E1 9998.261,E2 9998.261} C_VEL
LIN {X 0,Y 397.634,Z 955.186,A -85,B 0,C 180,E1 10005.78,E2 10005.78} C_VEL
LIN {X 0,Y 401.316,Z 917.733,A -85,B 0,C 180,E1 10012.012,E2 10012.012} C_VEL
LIN {X 0,Y 406.253,Z 870.749,A -85,B 0,C 180,E1 10016.451,E2 10016.451} C_VEL
LIN {X 0,Y 409.994,Z 816.866,A -85,B 0,C 180,E1 10018.891,E2 10018.891} C_VEL
LIN {X 0,Y 406.9,Z 792.819,A -85,B 0,C 180,E1 10019.557,E2 10019.557} C_VEL
LIN {X 0,Y 393.957,Z 754.81,A -85,B 0,C 180,E1 10021.336,E2 10021.336} C_VEL
LIN {X 0,Y 393.636,Z 754.81,A -85,B 0,C 180,E1 10032.43,E2 10032.43} C_VEL
LIN {X 0,Y 393.566,Z 754.81,A -85,B 0,C 180,E1 10043.301,E2 10043.301} C_VEL
LIN {X 0,Y 393.861,Z 754.81,A -85,B 0,C 180,E1 10053.702,E2 10053.702} C_VEL
LIN {X 0,Y 394.524,Z 754.81,A -85,B 0,C 180,E1 10065.524,E2 10065.524} C_VEL
LIN {X 0,Y 394.929,Z 754.81,A -85,B 0,C 180,E1 10076.699,E2 10076.699} C_VEL
LIN {X 0,Y 394.807,Z 754.81,A -85,B 0,C 180,E1 10085.517,E2 10085.517} C_VEL
LIN {X 0,Y 394.46,Z 754.81,A -85,B 0,C 180,E1 10096.773,E2 10096.773} C_VEL
LIN {X 0,Y 393.972,Z 754.81,A -85,B 0,C 180,E1 10106.297,E2 10106.297} C_VEL
LIN {X 0,Y 393.442,Z 754.81,A -85,B 0,C 180,E1 10117.746,E2 10117.746} C_VEL
LIN {X 0,Y 393.498,Z 754.81,A -85,B 0,C 180,E1 10128.771,E2 10128.771} C_VEL
LIN {X 0,Y 393.68,Z 754.81,A -85,B 0,C 180,E1 10140.155,E2 10140.155} C_VEL
LIN {X 0,Y 393.917,Z 754.81,A -85,B 0,C 180,E1 10150.884,E2 10150.884} C_VEL
LIN {X 0,Y 394.784,Z 754.81,A -85,B 0,C 180,E1 10162.267,E2 10162.267} C_VEL
LIN {X 0,Y 395.137,Z 756.551,A -85,B 0,C 180,E1 10169.724,E2 10169.724} C_VEL
LIN {X 0,Y 404.219,Z 799.197,A -85,B 0,C 180,E1 10172.647,E2 10172.647} C_VEL
LIN {X 0,Y 400.612,Z 835.152,A -85,B 0,C 180,E1 10176.798,E2 10176.798} C_VEL
LIN {X 0,Y 398.035,Z 858.532,A -85,B 0,C 180,E1 10182.104,E2 10182.104} C_VEL
LIN {X 0,Y 397.113,Z 867.986,A -85,B 0,C 180,E1 10186.655,E2 10186.655} C_VEL
LIN {X 0,Y 396.892,Z 870.065,A -85,B 0,C 180,E1 10191.299,E2 10191.299} C_VEL
LIN {X 0,Y 398.267,Z 860.374,A -85,B 0,C 180,E1 10197.852,E2 10197.852} C_VEL
LIN {X 0,Y 401.542,Z 837.06,A -85,B 0,C 180,E1 10203.477,E2 10203.477} C_VEL
LIN {X 0,Y 405.641,Z 802.15,A -85,B 0,C 180,E1 10207.684,E2 10207.684} C_VEL
LIN {X 0,Y 398.278,Z 767.296,A -85,B 0,C 180,E1 10210.541,E2 10210.541} C_VEL
LIN {X 0,Y 393.746,Z 754.81,A -85,B 0,C 180,E1 10211.506,E2 10211.506} C_VEL
LIN {X 0,Y 393.482,Z 754.81,A -85,B 0,C 180,E1 10222.244,E2 10222.244} C_VEL
LIN {X 0,Y 393.859,Z 754.81,A -85,B 0,C 180,E1 10233.695,E2 10233.695} C_VEL
LIN {X 0,Y 394.201,Z 754.81,A -85,B 0,C 180,E1 10245.506,E2 10245.506} C_VEL
LIN {X 0,Y 395.033,Z 754.81,A -85,B 0,C 180,E1 10256.694,E2 10256.694} C_VEL
LIN {X 0,Y 394.801,Z 754.81,A -85,B 0,C 180,E1 10267.729,E2 10267.729} C_VEL
LIN {X 0,Y 394.22,Z 754.81,A -85,B 0,C 180,E1 10279.096,E2 10279.096} C_VEL
LIN {X 0,Y 393.802,Z 754.81,A -85,B 0,C 180,E1 10289.881,E2 10289.881} C_VEL
LIN {X 0,Y 393.666,Z 754.81,A -85,B 0,C 180,E1 10301.261,E2 10301.261} C_VEL
LIN {X 0,Y 393.597,Z 754.81,A -85,B 0,C 180,E1 10312.218,E2 10312.218} C_VEL
LIN {X 0,Y 394.046,Z 756.395,A -85,B 0,C 180,E1 10318.295,E2 10318.295} C_VEL
LIN {X 0,Y 411.265,Z 806.215,A -85,B 0,C 180,E1 10320.551,E2 10320.551} C_VEL
LIN {X 0,Y 407.812,Z 859.868,A -85,B 0,C 180,E1 10322.582,E2 10322.582} C_VEL
LIN {X 0,Y 402.614,Z 908.427,A -85,B 0,C 180,E1 10326.686,E2 10326.686} C_VEL
LIN {X 0,Y 398.242,Z 948.306,A -85,B 0,C 180,E1 10332.694,E2 10332.694} C_VEL
LIN {X 0,Y 396.34,Z 975.755,A -85,B 0,C 180,E1 10340.079,E2 10340.079} C_VEL
LIN {X 0,Y 396.308,Z 985.239,A -85,B 0,C 180,E1 10345.053,E2 10345.053} C_VEL
LIN {X 0,Y 388.356,Z 987.04,A -85,B 0,C 180,E1 10350.099,E2 10350.099} C_VEL
LIN {X 0,Y 388.098,Z 980.553,A -85,B 0,C 180,E1 10357.302,E2 10357.302} C_VEL
LIN {X 0,Y 389.043,Z 959.667,A -85,B 0,C 180,E1 10364.689,E2 10364.689} C_VEL
LIN {X 0,Y 392.661,Z 923.893,A -85,B 0,C 180,E1 10371.393,E2 10371.393} C_VEL
LIN {X 0,Y 397.956,Z 877.456,A -85,B 0,C 180,E1 10376.306,E2 10376.306} C_VEL
LIN {X 0,Y 402.276,Z 824.719,A -85,B 0,C 180,E1 10379.086,E2 10379.086} C_VEL
LIN {X 0,Y 400.131,Z 796.385,A -85,B 0,C 180,E1 10379.888,E2 10379.888} C_VEL
LIN {X 0,Y 385.873,Z 754.81,A -85,B 0,C 180,E1 10381.741,E2 10381.741} C_VEL
LIN {X 0,Y 385.601,Z 754.81,A -85,B 0,C 180,E1 10393.531,E2 10393.531} C_VEL
LIN {X 0,Y 385.554,Z 754.81,A -85,B 0,C 180,E1 10405.203,E2 10405.203} C_VEL
LIN {X 0,Y 385.886,Z 754.81,A -85,B 0,C 180,E1 10415.614,E2 10415.614} C_VEL
LIN {X 0,Y 386.46,Z 754.81,A -85,B 0,C 180,E1 10425.215,E2 10425.215} C_VEL
LIN {X 0,Y 386.942,Z 754.81,A -85,B 0,C 180,E1 10436.63,E2 10436.63} C_VEL
LIN {X 0,Y 386.795,Z 754.81,A -85,B 0,C 180,E1 10445.632,E2 10445.632} C_VEL
LIN {X 0,Y 386.398,Z 754.81,A -85,B 0,C 180,E1 10457.134,E2 10457.134} C_VEL
LIN {X 0,Y 385.804,Z 754.81,A -85,B 0,C 180,E1 10467.741,E2 10467.741} C_VEL
LIN {X 0,Y 385.472,Z 754.81,A -85,B 0,C 180,E1 10479.851,E2 10479.851} C_VEL
LIN {X 0,Y 385.468,Z 754.81,A -85,B 0,C 180,E1 10490.152,E2 10490.152} C_VEL
LIN {X 0,Y 385.687,Z 754.81,A -85,B 0,C 180,E1 10500.537,E2 10500.537} C_VEL
LIN {X 0,Y 385.872,Z 754.81,A -85,B 0,C 180,E1 10510.47,E2 10510.47} C_VEL
LIN {X 0,Y 386.748,Z 754.81,A -85,B 0,C 180,E1 10522.105,E2 10522.105} C_VEL
LIN {X 0,Y 387.267,Z 756.214,A -85,B 0,C 180,E1 10529.22,E2 10529.22} C_VEL
LIN {X 0,Y 396.769,Z 799.189,A -85,B 0,C 180,E1 10532.21,E2 10532.21} C_VEL
LIN {X 0,Y 393.017,Z 835.232,A -85,B 0,C 180,E1 10536.373,E2 10536.373} C_VEL
LIN {X 0,Y 390.234,Z 859.126,A -85,B 0,C 180,E1 10541.78,E2 10541.78} C_VEL
LIN {X 0,Y 389.123,Z 869.764,A -85,B 0,C 180,E1 10547.151,E2 10547.151} C_VEL
LIN {X 0,Y 389.49,Z 869.104,A -85,B 0,C 180,E1 10554.148,E2 10554.148} C_VEL
LIN {X 0,Y 392.046,Z 853.63,A -85,B 0,C 180,E1 10560.534,E2 10560.534} C_VEL
LIN {X 0,Y 396.054,Z 825.206,A -85,B 0,C 180,E1 10565.769,E2 10565.769} C_VEL
LIN {X 0,Y 397.257,Z 790.368,A -85,B 0,C 180,E1 10569.293,E2 10569.293} C_VEL
LIN {X 0,Y 385.686,Z 754.81,A -85,B 0,C 180,E1 10572.207,E2 10572.207} C_VEL
LIN {X 0,Y 385.475,Z 754.81,A -85,B 0,C 180,E1 10583.809,E2 10583.809} C_VEL
LIN {X 0,Y 385.77,Z 754.81,A -85,B 0,C 180,E1 10593.1,E2 10593.1} C_VEL
LIN {X 0,Y 386.149,Z 754.81,A -85,B 0,C 180,E1 10605.197,E2 10605.197} C_VEL
LIN {X 0,Y 387.03,Z 754.81,A -85,B 0,C 180,E1 10616.625,E2 10616.625} C_VEL
LIN {X 0,Y 386.765,Z 754.81,A -85,B 0,C 180,E1 10627.89,E2 10627.89} C_VEL
LIN {X 0,Y 386.195,Z 754.81,A -85,B 0,C 180,E1 10639.509,E2 10639.509} C_VEL
LIN {X 0,Y 385.839,Z 754.81,A -85,B 0,C 180,E1 10649.445,E2 10649.445} C_VEL
LIN {X 0,Y 385.661,Z 754.81,A -85,B 0,C 180,E1 10660.482,E2 10660.482} C_VEL
LIN {X 0,Y 385.576,Z 754.81,A -85,B 0,C 180,E1 10670.124,E2 10670.124} C_VEL
LIN {X 0,Y 385.996,Z 756.415,A -85,B 0,C 180,E1 10677.614,E2 10677.614} C_VEL
LIN {X 0,Y 404.087,Z 806.071,A -85,B 0,C 180,E1 10680.037,E2 10680.037} C_VEL
LIN {X 0,Y 400.468,Z 859.833,A -85,B 0,C 180,E1 10682.133,E2 10682.133} C_VEL
LIN {X 0,Y 394.9,Z 908.366,A -85,B 0,C 180,E1 10686.363,E2 10686.363} C_VEL
LIN {X 0,Y 390.412,Z 946.56,A -85,B 0,C 180,E1 10692.227,E2 10692.227} C_VEL
LIN {X 0,Y 388.515,Z 973.124,A -85,B 0,C 180,E1 10699.308,E2 10699.308} C_VEL
LIN {X 0,Y 388.266,Z 985.781,A -85,B 0,C 180,E1 10706.64,E2 10706.64} C_VEL
LIN {X 0,Y 388.356,Z 987.04,A -85,B 0,C 180,E1 10710.099,E2 10710.099} C_VEL
LIN {X 0,Y 380.358,Z 982.676,A -85,B 0,C 180,E1 10715.242,E2 10715.242} C_VEL
LIN {X 0,Y 380.412,Z 966.392,A -85,B 0,C 180,E1 10722.675,E2 10722.675} C_VEL
LIN {X 0,Y 383.104,Z 935.915,A -85,B 0,C 180,E1 10729.677,E2 10729.677} C_VEL
LIN {X 0,Y 388.501,Z 892.927,A -85,B 0,C 180,E1 10735.294,E2 10735.294} C_VEL
LIN {X 0,Y 393.66,Z 842.438,A -85,B 0,C 180,E1 10738.809,E2 10738.809} C_VEL
LIN {X 0,Y 393.442,Z 800.442,A -85,B 0,C 180,E1 10740.21,E2 10740.21} C_VEL
LIN {X 0,Y 377.84,Z 754.81,A -85,B 0,C 180,E1 10742.101,E2 10742.101} C_VEL
LIN {X 0,Y 377.503,Z 754.81,A -85,B 0,C 180,E1 10751.958,E2 10751.958} C_VEL
LIN {X 0,Y 377.507,Z 754.81,A -85,B 0,C 180,E1 10761.62,E2 10761.62} C_VEL
LIN {X 0,Y 377.735,Z 754.81,A -85,B 0,C 180,E1 10772.486,E2 10772.486} C_VEL
LIN {X 0,Y 378.219,Z 754.81,A -85,B 0,C 180,E1 10782.49,E2 10782.49} C_VEL
LIN {X 0,Y 378.947,Z 754.81,A -85,B 0,C 180,E1 10794.257,E2 10794.257} C_VEL
LIN {X 0,Y 379.019,Z 754.81,A -85,B 0,C 180,E1 10803.446,E2 10803.446} C_VEL
LIN {X 0,Y 378.467,Z 754.81,A -85,B 0,C 180,E1 10815.111,E2 10815.111} C_VEL
LIN {X 0,Y 377.864,Z 754.81,A -85,B 0,C 180,E1 10825.357,E2 10825.357} C_VEL
LIN {X 0,Y 377.41,Z 754.81,A -85,B 0,C 180,E1 10835.668,E2 10835.668} C_VEL
LIN {X 0,Y 377.375,Z 754.81,A -85,B 0,C 180,E1 10845.271,E2 10845.271} C_VEL
LIN {X 0,Y 377.521,Z 754.81,A -85,B 0,C 180,E1 10857.133,E2 10857.133} C_VEL
LIN {X 0,Y 377.703,Z 754.81,A -85,B 0,C 180,E1 10867.56,E2 10867.56} C_VEL
LIN {X 0,Y 378.518,Z 754.81,A -85,B 0,C 180,E1 10879.605,E2 10879.605} C_VEL
LIN {X 0,Y 379.349,Z 755.935,A -85,B 0,C 180,E1 10888.695,E2 10888.695} C_VEL
LIN {X 0,Y 389.26,Z 799.657,A -85,B 0,C 180,E1 10891.797,E2 10891.797} C_VEL
LIN {X 0,Y 385.447,Z 835.256,A -85,B 0,C 180,E1 10895.931,E2 10895.931} C_VEL
LIN {X 0,Y 382.451,Z 859.681,A -85,B 0,C 180,E1 10901.443,E2 10901.443} C_VEL
LIN {X 0,Y 381.189,Z 871.185,A -85,B 0,C 180,E1 10907.372,E2 10907.372} C_VEL
LIN {X 0,Y 381.402,Z 871.511,A -85,B 0,C 180,E1 10913.117,E2 10913.117} C_VEL
LIN {X 0,Y 383.569,Z 858.941,A -85,B 0,C 180,E1 10919.64,E2 10919.64} C_VEL
LIN {X 0,Y 387.593,Z 832.997,A -85,B 0,C 180,E1 10925.238,E2 10925.238} C_VEL
LIN {X 0,Y 390.696,Z 795.565,A -85,B 0,C 180,E1 10929.423,E2 10929.423} C_VEL
LIN {X 0,Y 377.603,Z 754.81,A -85,B 0,C 180,E1 10932.937,E2 10932.937} C_VEL
LIN {X 0,Y 377.469,Z 754.81,A -85,B 0,C 180,E1 10944.338,E2 10944.338} C_VEL
LIN {X 0,Y 377.732,Z 754.81,A -85,B 0,C 180,E1 10955.046,E2 10955.046} C_VEL
LIN {X 0,Y 378.132,Z 754.81,A -85,B 0,C 180,E1 10964.876,E2 10964.876} C_VEL
LIN {X 0,Y 379.007,Z 754.81,A -85,B 0,C 180,E1 10976.554,E2 10976.554} C_VEL
LIN {X 0,Y 378.731,Z 754.81,A -85,B 0,C 180,E1 10988.059,E2 10988.059} C_VEL
LIN {X 0,Y 378.127,Z 754.81,A -85,B 0,C 180,E1 10999.943,E2 10999.943} C_VEL
LIN {X 0,Y 377.724,Z 754.81,A -85,B 0,C 180,E1 11010.255,E2 11010.255} C_VEL
LIN {X 0,Y 377.524,Z 754.81,A -85,B 0,C 180,E1 11021.957,E2 11021.957} C_VEL
LIN {X 0,Y 377.545,Z 754.81,A -85,B 0,C 180,E1 11031.606,E2 11031.606} C_VEL
LIN {X 0,Y 377.989,Z 756.612,A -85,B 0,C 180,E1 11036.906,E2 11036.906} C_VEL
LIN {X 0,Y 396.963,Z 809.107,A -85,B 0,C 180,E1 11039.578,E2 11039.578} C_VEL
LIN {X 0,Y 392.829,Z 862.483,A -85,B 0,C 180,E1 11041.834,E2 11041.834} C_VEL
LIN {X 0,Y 386.985,Z 910.338,A -85,B 0,C 180,E1 11046.26,E2 11046.26} C_VEL
LIN {X 0,Y 382.257,Z 949.289,A -85,B 0,C 180,E1 11052.678,E2 11052.678} C_VEL
LIN {X 0,Y 380.389,Z 974.821,A -85,B 0,C 180,E1 11060.239,E2 11060.239} C_VEL
LIN {X 0,Y 380.34,Z 984.608,A -85,B 0,C 180,E1 11066.569,E2 11066.569} C_VEL
LIN {X 0,Y 380.474,Z 984.571,A -85,B 0,C 180,E1 11073.431,E2 11073.431} C_VEL
LIN {X 0,Y 380.358,Z 982.676,A -85,B 0,C 180,E1 11075.242,E2 11075.242} C_VEL
LIN {X 0,Y 372.466,Z 972.403,A -85,B 0,C 180,E1 11080.292,E2 11080.292} C_VEL
LIN {X 0,Y 374.173,Z 946.606,A -85,B 0,C 180,E1 11087.71,E2 11087.71} C_VEL
LIN {X 0,Y 379.106,Z 906.86,A -85,B 0,C 180,E1 11094.068,E2 11094.068} C_VEL
LIN {X 0,Y 384.642,Z 858.602,A -85,B 0,C 180,E1 11098.34,E2 11098.34} C_VEL
LIN {X 0,Y 387.176,Z 805.895,A -85,B 0,C 180,E1 11100.483,E2 11100.483} C_VEL
LIN {X 0,Y 369.747,Z 754.81,A -85,B 0,C 180,E1 11102.719,E2 11102.719} C_VEL
LIN {X 0,Y 369.394,Z 754.81,A -85,B 0,C 180,E1 11114.038,E2 11114.038} C_VEL
LIN {X 0,Y 369.413,Z 754.81,A -85,B 0,C 180,E1 11123.444,E2 11123.444} C_VEL
LIN {X 0,Y 369.745,Z 754.81,A -85,B 0,C 180,E1 11134.475,E2 11134.475} C_VEL
LIN {X 0,Y 370.353,Z 754.81,A -85,B 0,C 180,E1 11144.556,E2 11144.556} C_VEL
LIN {X 0,Y 370.951,Z 754.81,A -85,B 0,C 180,E1 11156.485,E2 11156.485} C_VEL
LIN {X 0,Y 370.773,Z 754.81,A -85,B 0,C 180,E1 11165.876,E2 11165.876} C_VEL
LIN {X 0,Y 370.377,Z 754.81,A -85,B 0,C 180,E1 11175.657,E2 11175.657} C_VEL
LIN {X 0,Y 369.853,Z 754.81,A -85,B 0,C 180,E1 11185.523,E2 11185.523} C_VEL
LIN {X 0,Y 369.312,Z 754.81,A -85,B 0,C 180,E1 11196.745,E2 11196.745} C_VEL
LIN {X 0,Y 369.291,Z 754.81,A -85,B 0,C 180,E1 11207.307,E2 11207.307} C_VEL
LIN {X 0,Y 369.508,Z 754.81,A -85,B 0,C 180,E1 11219.11,E2 11219.11} C_VEL
LIN {X 0,Y 369.729,Z 754.81,A -85,B 0,C 180,E1 11229.58,E2 11229.58} C_VEL
LIN {X 0,Y 370.676,Z 754.81,A -85,B 0,C 180,E1 11241.761,E2 11241.761} C_VEL
LIN {X 0,Y 371.384,Z 756.601,A -85,B 0,C 180,E1 11248.184,E2 11248.184} C_VEL
LIN {X 0,Y 381.379,Z 799.501,A -85,B 0,C 180,E1 11251.287,E2 11251.287} C_VEL
LIN {X 0,Y 377.927,Z 835.263,A -85,B 0,C 180,E1 11255.472,E2 11255.472} C_VEL
LIN {X 0,Y 374.687,Z 860.231,A -85,B 0,C 180,E1 11261.091,E2 11261.091} C_VEL
LIN {X 0,Y 373.233,Z 872.679,A -85,B 0,C 180,E1 11267.754,E2 11267.754} C_VEL
LIN {X 0,Y 373.972,Z 870.523,A -85,B 0,C 180,E1 11275.219,E2 11275.219} C_VEL
LIN {X 0,Y 377.06,Z 853.608,A -85,B 0,C 180,E1 11281.782,E2 11281.782} C_VEL
LIN {X 0,Y 381.745,Z 824.389,A -85,B 0,C 180,E1 11287.031,E2 11287.031} C_VEL
LIN {X 0,Y 382.753,Z 794.101,A -85,B 0,C 180,E1 11290.224,E2 11290.224} C_VEL
LIN {X 0,Y 369.55,Z 754.81,A -85,B 0,C 180,E1 11293.763,E2 11293.763} C_VEL
LIN {X 0,Y 369.372,Z 754.81,A -85,B 0,C 180,E1 11303.432,E2 11303.432} C_VEL
LIN {X 0,Y 369.704,Z 754.81,A -85,B 0,C 180,E1 11314.466,E2 11314.466} C_VEL
LIN {X 0,Y 370.072,Z 754.81,A -85,B 0,C 180,E1 11324.538,E2 11324.538} C_VEL
LIN {X 0,Y 371,Z 754.81,A -85,B 0,C 180,E1 11336.479,E2 11336.479} C_VEL
LIN {X 0,Y 370.882,Z 754.81,A -85,B 0,C 180,E1 11345.868,E2 11345.868} C_VEL
LIN {X 0,Y 370.189,Z 754.81,A -85,B 0,C 180,E1 11357.903,E2 11357.903} C_VEL
LIN {X 0,Y 369.748,Z 754.81,A -85,B 0,C 180,E1 11368.16,E2 11368.16} C_VEL
LIN {X 0,Y 369.489,Z 754.81,A -85,B 0,C 180,E1 11379.536,E2 11379.536} C_VEL
LIN {X 0,Y 369.399,Z 754.81,A -85,B 0,C 180,E1 11390.449,E2 11390.449} C_VEL
LIN {X 0,Y 369.883,Z 756.545,A -85,B 0,C 180,E1 11396.134,E2 11396.134} C_VEL
LIN {X 0,Y 389.741,Z 808.975,A -85,B 0,C 180,E1 11399.011,E2 11399.011} C_VEL
LIN {X 0,Y 385.538,Z 862.147,A -85,B 0,C 180,E1 11401.333,E2 11401.333} C_VEL
LIN {X 0,Y 379.416,Z 909.441,A -85,B 0,C 180,E1 11405.797,E2 11405.797} C_VEL
LIN {X 0,Y 374.376,Z 948.091,A -85,B 0,C 180,E1 11412.302,E2 11412.302} C_VEL
LIN {X 0,Y 372.443,Z 973.651,A -85,B 0,C 180,E1 11420.028,E2 11420.028} C_VEL
LIN {X 0,Y 372.425,Z 983.55,A -85,B 0,C 180,E1 11426.628,E2 11426.628} C_VEL
LIN {X 0,Y 372.546,Z 983.22,A -85,B 0,C 180,E1 11433.675,E2 11433.675} C_VEL
LIN {X 0,Y 372.466,Z 972.403,A -85,B 0,C 180,E1 11440.292,E2 11440.292} C_VEL
LIN {X 0,Y 365.294,Z 957.214,A -85,B 0,C 180,E1 11445.151,E2 11445.151} C_VEL
LIN {X 0,Y 369.201,Z 922.783,A -85,B 0,C 180,E1 11452.143,E2 11452.143} C_VEL
LIN {X 0,Y 374.965,Z 878.069,A -85,B 0,C 180,E1 11457.298,E2 11457.298} C_VEL
LIN {X 0,Y 379.883,Z 826.258,A -85,B 0,C 180,E1 11460.321,E2 11460.321} C_VEL
LIN {X 0,Y 378.026,Z 801.847,A -85,B 0,C 180,E1 11461.155,E2 11461.155} C_VEL
LIN {X 0,Y 361.697,Z 754.81,A -85,B 0,C 180,E1 11463.464,E2 11463.464} C_VEL
LIN {X 0,Y 361.388,Z 754.81,A -85,B 0,C 180,E1 11473.86,E2 11473.86} C_VEL
LIN {X 0,Y 361.387,Z 754.81,A -85,B 0,C 180,E1 11485.47,E2 11485.47} C_VEL
LIN {X 0,Y 361.805,Z 754.81,A -85,B 0,C 180,E1 11496.521,E2 11496.521} C_VEL
LIN {X 0,Y 362.429,Z 754.81,A -85,B 0,C 180,E1 11506.689,E2 11506.689} C_VEL
LIN {X 0,Y 362.939,Z 754.81,A -85,B 0,C 180,E1 11516.407,E2 11516.407} C_VEL
LIN {X 0,Y 362.757,Z 754.81,A -85,B 0,C 180,E1 11526.006,E2 11526.006} C_VEL
LIN {X 0,Y 362.37,Z 754.81,A -85,B 0,C 180,E1 11535.799,E2 11535.799} C_VEL
LIN {X 0,Y 361.766,Z 754.81,A -85,B 0,C 180,E1 11546.136,E2 11546.136} C_VEL
LIN {X 0,Y 361.225,Z 754.81,A -85,B 0,C 180,E1 11557.533,E2 11557.533} C_VEL
LIN {X 0,Y 361.268,Z 754.81,A -85,B 0,C 180,E1 11569.374,E2 11569.374} C_VEL
LIN {X 0,Y 361.488,Z 754.81,A -85,B 0,C 180,E1 11581.132,E2 11581.132} C_VEL
LIN {X 0,Y 361.835,Z 754.81,A -85,B 0,C 180,E1 11591.665,E2 11591.665} C_VEL
LIN {X 0,Y 362.636,Z 754.81,A -85,B 0,C 180,E1 11601.577,E2 11601.577} C_VEL
LIN {X 0,Y 363.221,Z 756.142,A -85,B 0,C 180,E1 11607.605,E2 11607.605} C_VEL
LIN {X 0,Y 373.506,Z 799.563,A -85,B 0,C 180,E1 11610.776,E2 11610.776} C_VEL
LIN {X 0,Y 370.425,Z 835.271,A -85,B 0,C 180,E1 11614.994,E2 11614.994} C_VEL
LIN {X 0,Y 366.951,Z 860.774,A -85,B 0,C 180,E1 11620.725,E2 11620.725} C_VEL
LIN {X 0,Y 365.476,Z 872.668,A -85,B 0,C 180,E1 11626.513,E2 11626.513} C_VEL
LIN {X 0,Y 365.618,Z 874.013,A -85,B 0,C 180,E1 11633.223,E2 11633.223} C_VEL
LIN {X 0,Y 368.227,Z 861.349,A -85,B 0,C 180,E1 11640.211,E2 11640.211} C_VEL
LIN {X 0,Y 372.928,Z 834.848,A -85,B 0,C 180,E1 11646.16,E2 11646.16} C_VEL
LIN {X 0,Y 376.031,Z 798.281,A -85,B 0,C 180,E1 11650.468,E2 11650.468} C_VEL
LIN {X 0,Y 362.06,Z 757.834,A -85,B 0,C 180,E1 11654.217,E2 11654.217} C_VEL
LIN {X 0,Y 361.395,Z 754.81,A -85,B 0,C 180,E1 11654.743,E2 11654.743} C_VEL
LIN {X 0,Y 361.36,Z 754.81,A -85,B 0,C 180,E1 11665.459,E2 11665.459} C_VEL
LIN {X 0,Y 361.644,Z 754.81,A -85,B 0,C 180,E1 11676.503,E2 11676.503} C_VEL
LIN {X 0,Y 362.13,Z 754.81,A -85,B 0,C 180,E1 11686.671,E2 11686.671} C_VEL
LIN {X 0,Y 363.437,Z 754.81,A -85,B 0,C 180,E1 11698.801,E2 11698.801} C_VEL
LIN {X 0,Y 362.527,Z 754.81,A -85,B 0,C 180,E1 11710.855,E2 11710.855} C_VEL
LIN {X 0,Y 362.02,Z 754.81,A -85,B 0,C 180,E1 11720.871,E2 11720.871} C_VEL
LIN {X 0,Y 361.626,Z 754.81,A -85,B 0,C 180,E1 11731.635,E2 11731.635} C_VEL
LIN {X 0,Y 361.411,Z 754.81,A -85,B 0,C 180,E1 11743.85,E2 11743.85} C_VEL
LIN {X 0,Y 361.705,Z 756.001,A -85,B 0,C 180,E1 11755.294,E2 11755.294} C_VEL
LIN {X 0,Y 382.872,Z 811.625,A -85,B 0,C 180,E1 11758.518,E2 11758.518} C_VEL
LIN {X 0,Y 377.952,Z 864.97,A -85,B 0,C 180,E1 11761.032,E2 11761.032} C_VEL
LIN {X 0,Y 371.25,Z 912.673,A -85,B 0,C 180,E1 11765.873,E2 11765.873} C_VEL
LIN {X 0,Y 366.306,Z 949.644,A -85,B 0,C 180,E1 11772.556,E2 11772.556} C_VEL
LIN {X 0,Y 364.439,Z 973.738,A -85,B 0,C 180,E1 11780.413,E2 11780.413} C_VEL
LIN {X 0,Y 364.506,Z 982.277,A -85,B 0,C 180,E1 11786.42,E2 11786.42} C_VEL
LIN {X 0,Y 364.631,Z 982.137,A -85,B 0,C 180,E1 11793.58,E2 11793.58} C_VEL
LIN {X 0,Y 364.42,Z 968.994,A -85,B 0,C 180,E1 11801.349,E2 11801.349} C_VEL
LIN {X 0,Y 365.294,Z 957.214,A -85,B 0,C 180,E1 11805.151,E2 11805.151} C_VEL
LIN {X 0,Y 359.119,Z 937.531,A -85,B 0,C 180,E1 11809.731,E2 11809.731} C_VEL
LIN {X 0,Y 364.861,Z 896.133,A -85,B 0,C 180,E1 11815.896,E2 11815.896} C_VEL
LIN {X 0,Y 370.836,Z 846.695,A -85,B 0,C 180,E1 11819.863,E2 11819.863} C_VEL
LIN {X 0,Y 371.344,Z 805.612,A -85,B 0,C 180,E1 11821.503,E2 11821.503} C_VEL
LIN {X 0,Y 353.614,Z 754.81,A -85,B 0,C 180,E1 11823.991,E2 11823.991} C_VEL
LIN {X 0,Y 353.313,Z 754.81,A -85,B 0,C 180,E1 11835.132,E2 11835.132} C_VEL
LIN {X 0,Y 353.344,Z 754.81,A -85,B 0,C 180,E1 11846.879,E2 11846.879} C_VEL
LIN {X 0,Y 353.867,Z 754.81,A -85,B 0,C 180,E1 11858.625,E2 11858.625} C_VEL
LIN {X 0,Y 354.507,Z 754.81,A -85,B 0,C 180,E1 11868.897,E2 11868.897} C_VEL
LIN {X 0,Y 355.451,Z 754.81,A -85,B 0,C 180,E1 11881.226,E2 11881.226} C_VEL
LIN {X 0,Y 354.413,Z 754.81,A -85,B 0,C 180,E1 11893.624,E2 11893.624} C_VEL
LIN {X 0,Y 353.849,Z 754.81,A -85,B 0,C 180,E1 11904.047,E2 11904.047} C_VEL
LIN {X 0,Y 353.237,Z 754.81,A -85,B 0,C 180,E1 11915.453,E2 11915.453} C_VEL
LIN {X 0,Y 353.224,Z 754.81,A -85,B 0,C 180,E1 11925.149,E2 11925.149} C_VEL
LIN {X 0,Y 353.336,Z 754.81,A -85,B 0,C 180,E1 11937.528,E2 11937.528} C_VEL
LIN {X 0,Y 353.617,Z 754.81,A -85,B 0,C 180,E1 11948.605,E2 11948.605} C_VEL
LIN {X 0,Y 354.372,Z 754.81,A -85,B 0,C 180,E1 11958.888,E2 11958.888} C_VEL
LIN {X 0,Y 355.245,Z 756.474,A -85,B 0,C 180,E1 11967.032,E2 11967.032} C_VEL
LIN {X 0,Y 365.719,Z 799.976,A -85,B 0,C 180,E1 11970.293,E2 11970.293} C_VEL
LIN {X 0,Y 362.663,Z 837.018,A -85,B 0,C 180,E1 11974.8,E2 11974.8} C_VEL
LIN {X 0,Y 358.933,Z 863.107,A -85,B 0,C 180,E1 11980.967,E2 11980.967} C_VEL
LIN {X 0,Y 357.474,Z 874.6,A -85,B 0,C 180,E1 11987.211,E2 11987.211} C_VEL
LIN {X 0,Y 357.998,Z 874.409,A -85,B 0,C 180,E1 11994.295,E2 11994.295} C_VEL
LIN {X 0,Y 361.162,Z 860.216,A -85,B 0,C 180,E1 12001.274,E2 12001.274} C_VEL
LIN {X 0,Y 366.226,Z 832.587,A -85,B 0,C 180,E1 12007.148,E2 12007.148} C_VEL
LIN {X 0,Y 368.545,Z 798.951,A -85,B 0,C 180,E1 12011.109,E2 12011.109} C_VEL
LIN {X 0,Y 354.649,Z 759.124,A -85,B 0,C 180,E1 12014.968,E2 12014.968} C_VEL
LIN {X 0,Y 353.347,Z 754.81,A -85,B 0,C 180,E1 12015.649,E2 12015.649} C_VEL
LIN {X 0,Y 353.362,Z 754.81,A -85,B 0,C 180,E1 12027.529,E2 12027.529} C_VEL
LIN {X 0,Y 353.645,Z 754.81,A -85,B 0,C 180,E1 12038.605,E2 12038.605} C_VEL
LIN {X 0,Y 354.346,Z 754.81,A -85,B 0,C 180,E1 12048.885,E2 12048.885} C_VEL
LIN {X 0,Y 355.443,Z 754.81,A -85,B 0,C 180,E1 12058.774,E2 12058.774} C_VEL
LIN {X 0,Y 354.483,Z 754.81,A -85,B 0,C 180,E1 12071.104,E2 12071.104} C_VEL
LIN {X 0,Y 353.886,Z 754.81,A -85,B 0,C 180,E1 12082.784,E2 12082.784} C_VEL
LIN {X 0,Y 353.464,Z 754.81,A -85,B 0,C 180,E1 12093.154,E2 12093.154} C_VEL
LIN {X 0,Y 353.33,Z 754.81,A -85,B 0,C 180,E1 12105.123,E2 12105.123} C_VEL
LIN {X 0,Y 353.718,Z 756.594,A -85,B 0,C 180,E1 12114.453,E2 12114.453} C_VEL
LIN {X 0,Y 375.536,Z 811.624,A -85,B 0,C 180,E1 12117.893,E2 12117.893} C_VEL
LIN {X 0,Y 370.818,Z 863.786,A -85,B 0,C 180,E1 12120.419,E2 12120.419} C_VEL
LIN {X 0,Y 363.969,Z 910.452,A -85,B 0,C 180,E1 12125.194,E2 12125.194} C_VEL
LIN {X 0,Y 358.507,Z 947.794,A -85,B 0,C 180,E1 12131.989,E2 12131.989} C_VEL
LIN {X 0,Y 356.504,Z 972.593,A -85,B 0,C 180,E1 12140.197,E2 12140.197} C_VEL
LIN {X 0,Y 356.739,Z 982.237,A -85,B 0,C 180,E1 12148.425,E2 12148.425} C_VEL
LIN {X 0,Y 356.463,Z 978.28,A -85,B 0,C 180,E1 12156.111,E2 12156.111} C_VEL
LIN {X 0,Y 356.872,Z 960.253,A -85,B 0,C 180,E1 12164.154,E2 12164.154} C_VEL
LIN {X 0,Y 359.119,Z 937.531,A -85,B 0,C 180,E1 12169.731,E2 12169.731} C_VEL
LIN {X 0,Y 354.72,Z 913.86,A -85,B 0,C 180,E1 12173.93,E2 12173.93} C_VEL
LIN {X 0,Y 360.951,Z 867.6,A -85,B 0,C 180,E1 12178.915,E2 12178.915} C_VEL
LIN {X 0,Y 365.682,Z 814.46,A -85,B 0,C 180,E1 12181.637,E2 12181.637} C_VEL
LIN {X 0,Y 345.527,Z 754.81,A -85,B 0,C 180,E1 12184.613,E2 12184.613} C_VEL
LIN {X 0,Y 345.2,Z 754.81,A -85,B 0,C 180,E1 12197.051,E2 12197.051} C_VEL
LIN {X 0,Y 345.334,Z 754.81,A -85,B 0,C 180,E1 12208.975,E2 12208.975} C_VEL
LIN {X 0,Y 345.956,Z 754.81,A -85,B 0,C 180,E1 12220.796,E2 12220.796} C_VEL
LIN {X 0,Y 346.667,Z 754.81,A -85,B 0,C 180,E1 12231.19,E2 12231.19} C_VEL
LIN {X 0,Y 347.432,Z 754.81,A -85,B 0,C 180,E1 12241.255,E2 12241.255} C_VEL
LIN {X 0,Y 346.388,Z 754.81,A -85,B 0,C 180,E1 12253.946,E2 12253.946} C_VEL
LIN {X 0,Y 345.625,Z 754.81,A -85,B 0,C 180,E1 12265.825,E2 12265.825} C_VEL
LIN {X 0,Y 345.184,Z 754.81,A -85,B 0,C 180,E1 12276.41,E2 12276.41} C_VEL
LIN {X 0,Y 345.115,Z 754.81,A -85,B 0,C 180,E1 12287.032,E2 12287.032} C_VEL
LIN {X 0,Y 345.292,Z 754.81,A -85,B 0,C 180,E1 12298.99,E2 12298.99} C_VEL
LIN {X 0,Y 345.697,Z 754.81,A -85,B 0,C 180,E1 12310.776,E2 12310.776} C_VEL
LIN {X 0,Y 346.556,Z 754.81,A -85,B 0,C 180,E1 12321.183,E2 12321.183} C_VEL
LIN {X 0,Y 347.189,Z 756.563,A -85,B 0,C 180,E1 12326.426,E2 12326.426} C_VEL
LIN {X 0,Y 357.514,Z 798.03,A -85,B 0,C 180,E1 12329.555,E2 12329.555} C_VEL
LIN {X 0,Y 356.613,Z 827.959,A -85,B 0,C 180,E1 12332.931,E2 12332.931} C_VEL
LIN {X 0,Y 352.394,Z 857.388,A -85,B 0,C 180,E1 12338.668,E2 12338.668} C_VEL
LIN {X 0,Y 349.914,Z 873.257,A -85,B 0,C 180,E1 12345.082,E2 12345.082} C_VEL
LIN {X 0,Y 349.538,Z 877.269,A -85,B 0,C 180,E1 12351.656,E2 12351.656} C_VEL
LIN {X 0,Y 351.712,Z 868.191,A -85,B 0,C 180,E1 12359.143,E2 12359.143} C_VEL
LIN {X 0,Y 356.666,Z 844.809,A -85,B 0,C 180,E1 12365.732,E2 12365.732} C_VEL
LIN {X 0,Y 362.628,Z 809.492,A -85,B 0,C 180,E1 12370.637,E2 12370.637} C_VEL
LIN {X 0,Y 352.141,Z 771.035,A -85,B 0,C 180,E1 12374.758,E2 12374.758} C_VEL
LIN {X 0,Y 345.312,Z 754.81,A -85,B 0,C 180,E1 12376.479,E2 12376.479} C_VEL
LIN {X 0,Y 345.337,Z 754.81,A -85,B 0,C 180,E1 12388.971,E2 12388.971} C_VEL
LIN {X 0,Y 345.712,Z 754.81,A -85,B 0,C 180,E1 12400.775,E2 12400.775} C_VEL
LIN {X 0,Y 346.525,Z 754.81,A -85,B 0,C 180,E1 12411.18,E2 12411.18} C_VEL
LIN {X 0,Y 347.022,Z 754.81,A -85,B 0,C 180,E1 12421.25,E2 12421.25} C_VEL
LIN {X 0,Y 346.459,Z 754.81,A -85,B 0,C 180,E1 12431.365,E2 12431.365} C_VEL
LIN {X 0,Y 345.899,Z 754.81,A -85,B 0,C 180,E1 12441.892,E2 12441.892} C_VEL
LIN {X 0,Y 345.446,Z 754.81,A -85,B 0,C 180,E1 12453.303,E2 12453.303} C_VEL
LIN {X 0,Y 345.24,Z 754.81,A -85,B 0,C 180,E1 12463.508,E2 12463.508} C_VEL
LIN {X 0,Y 345.534,Z 756.302,A -85,B 0,C 180,E1 12473.5,E2 12473.5} C_VEL
LIN {X 0,Y 368.212,Z 811.831,A -85,B 0,C 180,E1 12477.243,E2 12477.243} C_VEL
LIN {X 0,Y 363.491,Z 864.556,A -85,B 0,C 180,E1 12479.935,E2 12479.935} C_VEL
LIN {X 0,Y 356.155,Z 911.541,A -85,B 0,C 180,E1 12484.949,E2 12484.949} C_VEL
LIN {X 0,Y 350.452,Z 948.637,A -85,B 0,C 180,E1 12492.07,E2 12492.07} C_VEL
LIN {X 0,Y 348.502,Z 972.702,A -85,B 0,C 180,E1 12500.603,E2 12500.603} C_VEL
LIN {X 0,Y 348.902,Z 981.138,A -85,B 0,C 180,E1 12508.755,E2 12508.755} C_VEL
LIN {X 0,Y 348.524,Z 977.002,A -85,B 0,C 180,E1 12516.25,E2 12516.25} C_VEL
LIN {X 0,Y 349.028,Z 958.781,A -85,B 0,C 180,E1 12524.479,E2 12524.479} C_VEL
LIN {X 0,Y 352.938,Z 925.715,A -85,B 0,C 180,E1 12532.058,E2 12532.058} C_VEL
LIN {X 0,Y 354.72,Z 913.86,A -85,B 0,C 180,E1 12533.93,E2 12533.93} C_VEL
LIN {X 0,Y 350.816,Z 886.707,A -85,B 0,C 180,E1 12537.586,E2 12537.586} C_VEL
LIN {X 0,Y 356.971,Z 835.89,A -85,B 0,C 180,E1 12541.316,E2 12541.316} C_VEL
LIN {X 0,Y 356.177,Z 807.458,A -85,B 0,C 180,E1 12542.498,E2 12542.498} C_VEL
LIN {X 0,Y 337.455,Z 754.81,A -85,B 0,C 180,E1 12545.289,E2 12545.289} C_VEL
LIN {X 0,Y 337.11,Z 754.81,A -85,B 0,C 180,E1 12557.97,E2 12557.97} C_VEL
LIN {X 0,Y 337.324,Z 754.81,A -85,B 0,C 180,E1 12568.849,E2 12568.849} C_VEL
LIN {X 0,Y 337.901,Z 754.81,A -85,B 0,C 180,E1 12580.319,E2 12580.319} C_VEL
LIN {X 0,Y 338.639,Z 754.81,A -85,B 0,C 180,E1 12590.979,E2 12590.979} C_VEL
LIN {X 0,Y 339.418,Z 754.81,A -85,B 0,C 180,E1 12601.284,E2 12601.284} C_VEL
LIN {X 0,Y 338.5,Z 754.81,A -85,B 0,C 180,E1 12611.642,E2 12611.642} C_VEL
LIN {X 0,Y 337.777,Z 754.81,A -85,B 0,C 180,E1 12622.921,E2 12622.921} C_VEL
LIN {X 0,Y 337.193,Z 754.81,A -85,B 0,C 180,E1 12634.237,E2 12634.237} C_VEL
LIN {X 0,Y 337.033,Z 754.81,A -85,B 0,C 180,E1 12645.738,E2 12645.738} C_VEL
LIN {X 0,Y 337.258,Z 754.81,A -85,B 0,C 180,E1 12656.356,E2 12656.356} C_VEL
LIN {X 0,Y 337.502,Z 754.81,A -85,B 0,C 180,E1 12667.529,E2 12667.529} C_VEL
LIN {X 0,Y 338.262,Z 754.81,A -85,B 0,C 180,E1 12678.352,E2 12678.352} C_VEL
LIN {X 0,Y 339.054,Z 756.606,A -85,B 0,C 180,E1 12685.788,E2 12685.788} C_VEL
LIN {X 0,Y 349.609,Z 797.55,A -85,B 0,C 180,E1 12688.933,E2 12688.933} C_VEL
LIN {X 0,Y 349.871,Z 822.952,A -85,B 0,C 180,E1 12691.744,E2 12691.744} C_VEL
LIN {X 0,Y 345.153,Z 854.89,A -85,B 0,C 180,E1 12697.469,E2 12697.469} C_VEL
LIN {X 0,Y 342.242,Z 873.001,A -85,B 0,C 180,E1 12704.115,E2 12704.115} C_VEL
LIN {X 0,Y 341.735,Z 878.33,A -85,B 0,C 180,E1 12712.176,E2 12712.176} C_VEL
LIN {X 0,Y 344.193,Z 868.728,A -85,B 0,C 180,E1 12719.736,E2 12719.736} C_VEL
LIN {X 0,Y 349.568,Z 844.964,A -85,B 0,C 180,E1 12726.409,E2 12726.409} C_VEL
LIN {X 0,Y 355.364,Z 808.883,A -85,B 0,C 180,E1 12731.446,E2 12731.446} C_VEL
LIN {X 0,Y 343.417,Z 769.01,A -85,B 0,C 180,E1 12735.886,E2 12735.886} C_VEL
LIN {X 0,Y 337.178,Z 754.81,A -85,B 0,C 180,E1 12737.497,E2 12737.497} C_VEL
LIN {X 0,Y 337.326,Z 754.81,A -85,B 0,C 180,E1 12748.841,E2 12748.841} C_VEL
LIN {X 0,Y 337.662,Z 754.81,A -85,B 0,C 180,E1 12760.298,E2 12760.298} C_VEL
LIN {X 0,Y 338.503,Z 754.81,A -85,B 0,C 180,E1 12770.969,E2 12770.969} C_VEL
LIN {X 0,Y 339.028,Z 754.81,A -85,B 0,C 180,E1 12781.279,E2 12781.279} C_VEL
LIN {X 0,Y 338.409,Z 754.81,A -85,B 0,C 180,E1 12791.639,E2 12791.639} C_VEL
LIN {X 0,Y 337.763,Z 754.81,A -85,B 0,C 180,E1 12802.919,E2 12802.919} C_VEL
LIN {X 0,Y 337.379,Z 754.81,A -85,B 0,C 180,E1 12814.208,E2 12814.208} C_VEL
LIN {X 0,Y 337.15,Z 754.81,A -85,B 0,C 180,E1 12825.76,E2 12825.76} C_VEL
LIN {X 0,Y 337.449,Z 755.987,A -85,B 0,C 180,E1 12832.498,E2 12832.498} C_VEL
LIN {X 0,Y 360.819,Z 811.671,A -85,B 0,C 180,E1 12836.529,E2 12836.529} C_VEL
LIN {X 0,Y 356.497,Z 863.468,A -85,B 0,C 180,E1 12839.282,E2 12839.282} C_VEL
LIN {X 0,Y 348.76,Z 910.461,A -85,B 0,C 180,E1 12844.38,E2 12844.38} C_VEL
LIN {X 0,Y 342.62,Z 947.323,A -85,B 0,C 180,E1 12851.589,E2 12851.589} C_VEL
LIN {X 0,Y 340.545,Z 971.561,A -85,B 0,C 180,E1 12860.381,E2 12860.381} C_VEL
LIN {X 0,Y 340.99,Z 979.958,A -85,B 0,C 180,E1 12868.726,E2 12868.726} C_VEL
LIN {X 0,Y 340.589,Z 975.723,A -85,B 0,C 180,E1 12876.396,E2 12876.396} C_VEL
LIN {X 0,Y 341.172,Z 957.305,A -85,B 0,C 180,E1 12884.82,E2 12884.82} C_VEL
LIN {X 0,Y 345.287,Z 924.361,A -85,B 0,C 180,E1 12892.482,E2 12892.482} C_VEL
LIN {X 0,Y 350.816,Z 886.707,A -85,B 0,C 180,E1 12897.586,E2 12897.586} C_VEL
LIN {X 0,Y 347.288,Z 856.51,A -85,B 0,C 180,E1 12900.591,E2 12900.591} C_VEL
LIN {X 0,Y 349.41,Z 811.075,A -85,B 0,C 180,E1 12902.883,E2 12902.883} C_VEL
LIN {X 0,Y 329.457,Z 754.81,A -85,B 0,C 180,E1 12905.862,E2 12905.862} C_VEL
LIN {X 0,Y 329.107,Z 754.81,A -85,B 0,C 180,E1 12918.045,E2 12918.045} C_VEL
LIN {X 0,Y 329.312,Z 754.81,A -85,B 0,C 180,E1 12928.491,E2 12928.491} C_VEL
LIN {X 0,Y 329.889,Z 754.81,A -85,B 0,C 180,E1 12940.573,E2 12940.573} C_VEL
LIN {X 0,Y 330.798,Z 754.81,A -85,B 0,C 180,E1 12953.418,E2 12953.418} C_VEL
LIN {X 0,Y 330.91,Z 754.81,A -85,B 0,C 180,E1 12963.948,E2 12963.948} C_VEL
LIN {X 0,Y 330.306,Z 754.81,A -85,B 0,C 180,E1 12974.64,E2 12974.64} C_VEL
LIN {X 0,Y 329.547,Z 754.81,A -85,B 0,C 180,E1 12986.104,E2 12986.104} C_VEL
LIN {X 0,Y 328.999,Z 754.81,A -85,B 0,C 180,E1 12998.518,E2 12998.518} C_VEL
LIN {X 0,Y 328.993,Z 754.81,A -85,B 0,C 180,E1 13009.566,E2 13009.566} C_VEL
LIN {X 0,Y 329.299,Z 754.81,A -85,B 0,C 180,E1 13021.059,E2 13021.059} C_VEL
LIN {X 0,Y 329.75,Z 754.81,A -85,B 0,C 180,E1 13032.593,E2 13032.593} C_VEL
LIN {X 0,Y 330.803,Z 755.339,A -85,B 0,C 180,E1 13045.065,E2 13045.065} C_VEL
LIN {X 0,Y 341.636,Z 796.048,A -85,B 0,C 180,E1 13048.201,E2 13048.201} C_VEL
LIN {X 0,Y 342.539,Z 822.156,A -85,B 0,C 180,E1 13051.11,E2 13051.11} C_VEL
LIN {X 0,Y 337.563,Z 854.525,A -85,B 0,C 180,E1 13056.822,E2 13056.822} C_VEL
LIN {X 0,Y 334.491,Z 873.298,A -85,B 0,C 180,E1 13063.539,E2 13063.539} C_VEL
LIN {X 0,Y 333.71,Z 879.722,A -85,B 0,C 180,E1 13071.204,E2 13071.204} C_VEL
LIN {X 0,Y 335.948,Z 872.092,A -85,B 0,C 180,E1 13079.051,E2 13079.051} C_VEL
LIN {X 0,Y 341.356,Z 849.998,A -85,B 0,C 180,E1 13086.108,E2 13086.108} C_VEL
LIN {X 0,Y 348.162,Z 815.187,A -85,B 0,C 180,E1 13091.469,E2 13091.469} C_VEL
LIN {X 0,Y 339.612,Z 778.614,A -85,B 0,C 180,E1 13095.824,E2 13095.824} C_VEL
LIN {X 0,Y 329.101,Z 754.81,A -85,B 0,C 180,E1 13098.442,E2 13098.442} C_VEL
LIN {X 0,Y 329.355,Z 754.81,A -85,B 0,C 180,E1 13111.062,E2 13111.062} C_VEL
LIN {X 0,Y 329.746,Z 754.81,A -85,B 0,C 180,E1 13122.59,E2 13122.59} C_VEL
LIN {X 0,Y 330.598,Z 754.81,A -85,B 0,C 180,E1 13133.407,E2 13133.407} C_VEL
LIN {X 0,Y 331.019,Z 754.81,A -85,B 0,C 180,E1 13141.31,E2 13141.31} C_VEL
LIN {X 0,Y 330.363,Z 754.81,A -85,B 0,C 180,E1 13151.926,E2 13151.926} C_VEL
LIN {X 0,Y 329.761,Z 754.81,A -85,B 0,C 180,E1 13163.023,E2 13163.023} C_VEL
LIN {X 0,Y 329.236,Z 754.81,A -85,B 0,C 180,E1 13175.177,E2 13175.177} C_VEL
LIN {X 0,Y 329.141,Z 754.81,A -85,B 0,C 180,E1 13185.61,E2 13185.61} C_VEL
LIN {X 0,Y 329.514,Z 756.715,A -85,B 0,C 180,E1 13191.474,E2 13191.474} C_VEL
LIN {X 0,Y 353.349,Z 811.201,A -85,B 0,C 180,E1 13195.76,E2 13195.76} C_VEL
LIN {X 0,Y 351.751,Z 848.47,A -85,B 0,C 180,E1 13197.64,E2 13197.64} C_VEL
LIN {X 0,Y 343.75,Z 896.886,A -85,B 0,C 180,E1 13202.057,E2 13202.057} C_VEL
LIN {X 0,Y 336.087,Z 936.878,A -85,B 0,C 180,E1 13208.825,E2 13208.825} C_VEL
LIN {X 0,Y 332.711,Z 963.45,A -85,B 0,C 180,E1 13216.818,E2 13216.818} C_VEL
LIN {X 0,Y 332.771,Z 976.619,A -85,B 0,C 180,E1 13224.768,E2 13224.768} C_VEL
LIN {X 0,Y 332.99,Z 978.647,A -85,B 0,C 180,E1 13231.307,E2 13231.307} C_VEL
LIN {X 0,Y 332.722,Z 970.384,A -85,B 0,C 180,E1 13239.187,E2 13239.187} C_VEL
LIN {X 0,Y 334.265,Z 946.109,A -85,B 0,C 180,E1 13247.977,E2 13247.977} C_VEL
LIN {X 0,Y 339.921,Z 908.263,A -85,B 0,C 180,E1 13255.273,E2 13255.273} C_VEL
LIN {X 0,Y 346.617,Z 861.585,A -85,B 0,C 180,E1 13260.233,E2 13260.233} C_VEL
LIN {X 0,Y 347.288,Z 856.51,A -85,B 0,C 180,E1 13260.591,E2 13260.591} C_VEL
LIN {X 0,Y 343.174,Z 823.944,A -85,B 0,C 180,E1 13262.841,E2 13262.841} C_VEL
LIN {X 0,Y 331.169,Z 781.086,A -85,B 0,C 180,E1 13265.022,E2 13265.022} C_VEL
LIN {X 0,Y 321.314,Z 754.81,A -85,B 0,C 180,E1 13266.691,E2 13266.691} C_VEL
LIN {X 0,Y 321.057,Z 754.81,A -85,B 0,C 180,E1 13277.111,E2 13277.111} C_VEL
LIN {X 0,Y 321.131,Z 754.81,A -85,B 0,C 180,E1 13287.085,E2 13287.085} C_VEL
LIN {X 0,Y 321.723,Z 754.81,A -85,B 0,C 180,E1 13299.286,E2 13299.286} C_VEL
LIN {X 0,Y 322.586,Z 754.81,A -85,B 0,C 180,E1 13310.527,E2 13310.527} C_VEL
LIN {X 0,Y 323.385,Z 754.81,A -85,B 0,C 180,E1 13321.348,E2 13321.348} C_VEL
LIN {X 0,Y 322.391,Z 754.81,A -85,B 0,C 180,E1 13332.233,E2 13332.233} C_VEL
LIN {X 0,Y 321.653,Z 754.81,A -85,B 0,C 180,E1 13343.646,E2 13343.646} C_VEL
LIN {X 0,Y 321.013,Z 754.81,A -85,B 0,C 180,E1 13356.227,E2 13356.227} C_VEL
LIN {X 0,Y 320.962,Z 754.81,A -85,B 0,C 180,E1 13367.132,E2 13367.132} C_VEL
LIN {X 0,Y 321.073,Z 754.81,A -85,B 0,C 180,E1 13377.073,E2 13377.073} C_VEL
LIN {X 0,Y 321.5,Z 754.81,A -85,B 0,C 180,E1 13389.266,E2 13389.266} C_VEL
LIN {X 0,Y 322.439,Z 754.81,A -85,B 0,C 180,E1 13400.518,E2 13400.518} C_VEL
LIN {X 0,Y 322.798,Z 756.164,A -85,B 0,C 180,E1 13404.392,E2 13404.392} C_VEL
LIN {X 0,Y 333.895,Z 795.957,A -85,B 0,C 180,E1 13407.585,E2 13407.585} C_VEL
LIN {X 0,Y 335.084,Z 822.745,A -85,B 0,C 180,E1 13410.637,E2 13410.637} C_VEL
LIN {X 0,Y 329.923,Z 854.514,A -85,B 0,C 180,E1 13416.271,E2 13416.271} C_VEL
LIN {X 0,Y 326.667,Z 874.003,A -85,B 0,C 180,E1 13423.19,E2 13423.19} C_VEL
LIN {X 0,Y 325.723,Z 880.891,A -85,B 0,C 180,E1 13430.452,E2 13430.452} C_VEL
LIN {X 0,Y 327.856,Z 874.699,A -85,B 0,C 180,E1 13438.618,E2 13438.618} C_VEL
LIN {X 0,Y 333.269,Z 854.392,A -85,B 0,C 180,E1 13445.861,E2 13445.861} C_VEL
LIN {X 0,Y 340.392,Z 821.172,A -85,B 0,C 180,E1 13451.539,E2 13451.539} C_VEL
LIN {X 0,Y 336.788,Z 792.883,A -85,B 0,C 180,E1 13455.13,E2 13455.13} C_VEL
LIN {X 0,Y 321.036,Z 754.81,A -85,B 0,C 180,E1 13459.841,E2 13459.841} C_VEL
LIN {X 0,Y 321.343,Z 754.81,A -85,B 0,C 180,E1 13470.888,E2 13470.888} C_VEL
LIN {X 0,Y 321.713,Z 754.81,A -85,B 0,C 180,E1 13482.141,E2 13482.141} C_VEL
LIN {X 0,Y 322.568,Z 754.81,A -85,B 0,C 180,E1 13493.242,E2 13493.242} C_VEL
LIN {X 0,Y 323.026,Z 754.81,A -85,B 0,C 180,E1 13501.343,E2 13501.343} C_VEL
LIN {X 0,Y 322.309,Z 754.81,A -85,B 0,C 180,E1 13512.229,E2 13512.229} C_VEL
LIN {X 0,Y 321.65,Z 754.81,A -85,B 0,C 180,E1 13523.639,E2 13523.639} C_VEL
LIN {X 0,Y 321.21,Z 754.81,A -85,B 0,C 180,E1 13536.192,E2 13536.192} C_VEL
LIN {X 0,Y 321.098,Z 754.81,A -85,B 0,C 180,E1 13547.095,E2 13547.095} C_VEL
LIN {X 0,Y 321.44,Z 756.833,A -85,B 0,C 180,E1 13550.327,E2 13550.327} C_VEL
LIN {X 0,Y 345.855,Z 810.65,A -85,B 0,C 180,E1 13554.939,E2 13554.939} C_VEL
LIN {X 0,Y 346.918,Z 831.65,A -85,B 0,C 180,E1 13556.051,E2 13556.051} C_VEL
LIN {X 0,Y 339.201,Z 882.041,A -85,B 0,C 180,E1 13559.782,E2 13559.782} C_VEL
LIN {X 0,Y 330.786,Z 924.294,A -85,B 0,C 180,E1 13565.878,E2 13565.878} C_VEL
LIN {X 0,Y 325.611,Z 955.27,A -85,B 0,C 180,E1 13573.776,E2 13573.776} C_VEL
LIN {X 0,Y 324.58,Z 972.393,A -85,B 0,C 180,E1 13581.938,E2 13581.938} C_VEL
LIN {X 0,Y 325.135,Z 977.595,A -85,B 0,C 180,E1 13588.664,E2 13588.664} C_VEL
LIN {X 0,Y 324.719,Z 973.15,A -85,B 0,C 180,E1 13596.71,E2 13596.71} C_VEL
LIN {X 0,Y 325.688,Z 953.36,A -85,B 0,C 180,E1 13605.853,E2 13605.853} C_VEL
LIN {X 0,Y 330.383,Z 918.85,A -85,B 0,C 180,E1 13613.882,E2 13613.882} C_VEL
LIN {X 0,Y 337.445,Z 873.816,A -85,B 0,C 180,E1 13619.651,E2 13619.651} C_VEL
LIN {X 0,Y 343.174,Z 823.944,A -85,B 0,C 180,E1 13622.841,E2 13622.841} C_VEL
LIN {X 0,Y 331.775,Z 804.945,A -85,B 0,C 180,E1 13624.408,E2 13624.408} C_VEL
LIN {X 0,Y 313.256,Z 754.81,A -85,B 0,C 180,E1 13627.271,E2 13627.271} C_VEL
LIN {X 0,Y 312.934,Z 754.81,A -85,B 0,C 180,E1 13639.11,E2 13639.11} C_VEL
LIN {X 0,Y 313.149,Z 754.81,A -85,B 0,C 180,E1 13649.418,E2 13649.418} C_VEL
LIN {X 0,Y 313.847,Z 754.81,A -85,B 0,C 180,E1 13661.685,E2 13661.685} C_VEL
LIN {X 0,Y 314.725,Z 754.81,A -85,B 0,C 180,E1 13673.08,E2 13673.08} C_VEL
LIN {X 0,Y 314.857,Z 754.81,A -85,B 0,C 180,E1 13684.149,E2 13684.149} C_VEL
LIN {X 0,Y 314.185,Z 754.81,A -85,B 0,C 180,E1 13695.41,E2 13695.41} C_VEL
LIN {X 0,Y 313.391,Z 754.81,A -85,B 0,C 180,E1 13707.393,E2 13707.393} C_VEL
LIN {X 0,Y 312.945,Z 754.81,A -85,B 0,C 180,E1 13717.316,E2 13717.316} C_VEL
LIN {X 0,Y 312.854,Z 754.81,A -85,B 0,C 180,E1 13729.091,E2 13729.091} C_VEL
LIN {X 0,Y 313.101,Z 754.81,A -85,B 0,C 180,E1 13739.407,E2 13739.407} C_VEL
LIN {X 0,Y 313.618,Z 754.81,A -85,B 0,C 180,E1 13751.667,E2 13751.667} C_VEL
LIN {X 0,Y 314.901,Z 756.823,A -85,B 0,C 180,E1 13763.699,E2 13763.699} C_VEL
LIN {X 0,Y 326.206,Z 795.832,A -85,B 0,C 180,E1 13766.939,E2 13766.939} C_VEL
LIN {X 0,Y 327.514,Z 824.153,A -85,B 0,C 180,E1 13770.246,E2 13770.246} C_VEL
LIN {X 0,Y 322.126,Z 856.031,A -85,B 0,C 180,E1 13776.084,E2 13776.084} C_VEL
LIN {X 0,Y 318.582,Z 876.415,A -85,B 0,C 180,E1 13783.825,E2 13783.825} C_VEL
LIN {X 0,Y 317.921,Z 882.111,A -85,B 0,C 180,E1 13791.43,E2 13791.43} C_VEL
LIN {X 0,Y 320.605,Z 874.347,A -85,B 0,C 180,E1 13799.802,E2 13799.802} C_VEL
LIN {X 0,Y 326.914,Z 851.598,A -85,B 0,C 180,E1 13807.322,E2 13807.322} C_VEL
LIN {X 0,Y 334.287,Z 816.143,A -85,B 0,C 180,E1 13812.945,E2 13812.945} C_VEL
LIN {X 0,Y 323.493,Z 777.227,A -85,B 0,C 180,E1 13818.062,E2 13818.062} C_VEL
LIN {X 0,Y 313.027,Z 754.81,A -85,B 0,C 180,E1 13820.808,E2 13820.808} C_VEL
LIN {X 0,Y 313.349,Z 754.81,A -85,B 0,C 180,E1 13833.631,E2 13833.631} C_VEL
LIN {X 0,Y 313.82,Z 754.81,A -85,B 0,C 180,E1 13844.572,E2 13844.572} C_VEL
LIN {X 0,Y 314.827,Z 754.81,A -85,B 0,C 180,E1 13855.85,E2 13855.85} C_VEL
LIN {X 0,Y 314.67,Z 754.81,A -85,B 0,C 180,E1 13866.921,E2 13866.921} C_VEL
LIN {X 0,Y 313.798,Z 754.81,A -85,B 0,C 180,E1 13879.433,E2 13879.433} C_VEL
LIN {X 0,Y 313.179,Z 754.81,A -85,B 0,C 180,E1 13892.007,E2 13892.007} C_VEL
LIN {X 0,Y 312.963,Z 754.81,A -85,B 0,C 180,E1 13904.671,E2 13904.671} C_VEL
LIN {X 0,Y 313.347,Z 756.769,A -85,B 0,C 180,E1 13909.091,E2 13909.091} C_VEL
LIN {X 0,Y 338.134,Z 809.348,A -85,B 0,C 180,E1 13914.003,E2 13914.003} C_VEL
LIN {X 0,Y 340.333,Z 830.163,A -85,B 0,C 180,E1 13915.268,E2 13915.268} C_VEL
LIN {X 0,Y 332.476,Z 879.508,A -85,B 0,C 180,E1 13918.913,E2 13918.913} C_VEL
LIN {X 0,Y 323.591,Z 922.018,A -85,B 0,C 180,E1 13925.035,E2 13925.035} C_VEL
LIN {X 0,Y 317.742,Z 954.481,A -85,B 0,C 180,E1 13933.475,E2 13933.475} C_VEL
LIN {X 0,Y 316.742,Z 972.948,A -85,B 0,C 180,E1 13943.121,E2 13943.121} C_VEL
LIN {X 0,Y 317.165,Z 976.215,A -85,B 0,C 180,E1 13951.372,E2 13951.372} C_VEL
LIN {X 0,Y 316.731,Z 966.605,A -85,B 0,C 180,E1 13960.232,E2 13960.232} C_VEL
LIN {X 0,Y 318.674,Z 942.01,A -85,B 0,C 180,E1 13969.112,E2 13969.112} C_VEL
LIN {X 0,Y 324.841,Z 905.154,A -85,B 0,C 180,E1 13976.349,E2 13976.349} C_VEL
LIN {X 0,Y 332.094,Z 858.214,A -85,B 0,C 180,E1 13981.416,E2 13981.416} C_VEL
LIN {X 0,Y 334.521,Z 813.987,A -85,B 0,C 180,E1 13983.893,E2 13983.893} C_VEL
LIN {X 0,Y 331.775,Z 804.945,A -85,B 0,C 180,E1 13984.408,E2 13984.408} C_VEL
LIN {X 0,Y 313.769,Z 776.957,A -85,B 0,C 180,E1 13986.648,E2 13986.648} C_VEL
LIN {X 0,Y 305.031,Z 754.81,A -85,B 0,C 180,E1 13988.456,E2 13988.456} C_VEL
LIN {X 0,Y 304.855,Z 754.81,A -85,B 0,C 180,E1 14001.525,E2 14001.525} C_VEL
LIN {X 0,Y 305.203,Z 754.81,A -85,B 0,C 180,E1 14011.816,E2 14011.816} C_VEL
LIN {X 0,Y 306.037,Z 754.81,A -85,B 0,C 180,E1 14024.177,E2 14024.177} C_VEL
LIN {X 0,Y 306.848,Z 754.81,A -85,B 0,C 180,E1 14035.749,E2 14035.749} C_VEL
LIN {X 0,Y 306.842,Z 754.81,A -85,B 0,C 180,E1 14044.258,E2 14044.258} C_VEL
LIN {X 0,Y 306.114,Z 754.81,A -85,B 0,C 180,E1 14055.826,E2 14055.826} C_VEL
LIN {X 0,Y 305.234,Z 754.81,A -85,B 0,C 180,E1 14068.189,E2 14068.189} C_VEL
LIN {X 0,Y 304.759,Z 754.81,A -85,B 0,C 180,E1 14079.48,E2 14079.48} C_VEL
LIN {X 0,Y 304.794,Z 754.81,A -85,B 0,C 180,E1 14091.509,E2 14091.509} C_VEL
LIN {X 0,Y 305.108,Z 754.81,A -85,B 0,C 180,E1 14101.801,E2 14101.801} C_VEL
LIN {X 0,Y 305.766,Z 754.81,A -85,B 0,C 180,E1 14114.158,E2 14114.158} C_VEL
LIN {X 0,Y 306.672,Z 756.242,A -85,B 0,C 180,E1 14122.893,E2 14122.893} C_VEL
LIN {X 0,Y 318.684,Z 796.791,A -85,B 0,C 180,E1 14126.375,E2 14126.375} C_VEL
LIN {X 0,Y 320.125,Z 824.358,A -85,B 0,C 180,E1 14129.677,E2 14129.677} C_VEL
LIN {X 0,Y 314.337,Z 857.547,A -85,B 0,C 180,E1 14135.888,E2 14135.888} C_VEL
LIN {X 0,Y 310.786,Z 877.046,A -85,B 0,C 180,E1 14143.411,E2 14143.411} C_VEL
LIN {X 0,Y 310.046,Z 883.3,A -85,B 0,C 180,E1 14151.536,E2 14151.536} C_VEL
LIN {X 0,Y 312.855,Z 875.848,A -85,B 0,C 180,E1 14160.007,E2 14160.007} C_VEL
LIN {X 0,Y 319.374,Z 853.87,A -85,B 0,C 180,E1 14167.629,E2 14167.629} C_VEL
LIN {X 0,Y 327.254,Z 819.978,A -85,B 0,C 180,E1 14173.298,E2 14173.298} C_VEL
LIN {X 0,Y 318.104,Z 782.82,A -85,B 0,C 180,E1 14178.473,E2 14178.473} C_VEL
LIN {X 0,Y 304.991,Z 754.81,A -85,B 0,C 180,E1 14182.087,E2 14182.087} C_VEL
LIN {X 0,Y 305.306,Z 754.81,A -85,B 0,C 180,E1 14195.004,E2 14195.004} C_VEL
LIN {X 0,Y 305.998,Z 754.81,A -85,B 0,C 180,E1 14207.101,E2 14207.101} C_VEL
LIN {X 0,Y 307.328,Z 754.81,A -85,B 0,C 180,E1 14218.582,E2 14218.582} C_VEL
LIN {X 0,Y 306.384,Z 754.81,A -85,B 0,C 180,E1 14229.979,E2 14229.979} C_VEL
LIN {X 0,Y 305.634,Z 754.81,A -85,B 0,C 180,E1 14241.859,E2 14241.859} C_VEL
LIN {X 0,Y 305.108,Z 754.81,A -85,B 0,C 180,E1 14254.885,E2 14254.885} C_VEL
LIN {X 0,Y 305.177,Z 756.789,A -85,B 0,C 180,E1 14267.733,E2 14267.733} C_VEL
LIN {X 0,Y 330.515,Z 808.64,A -85,B 0,C 180,E1 14273.048,E2 14273.048} C_VEL
LIN {X 0,Y 333.788,Z 828.697,A -85,B 0,C 180,E1 14274.445,E2 14274.445} C_VEL
LIN {X 0,Y 325.539,Z 878.65,A -85,B 0,C 180,E1 14278.174,E2 14278.174} C_VEL
LIN {X 0,Y 316.188,Z 921.031,A -85,B 0,C 180,E1 14284.409,E2 14284.409} C_VEL
LIN {X 0,Y 310.077,Z 952.678,A -85,B 0,C 180,E1 14292.771,E2 14292.771} C_VEL
LIN {X 0,Y 308.699,Z 970.128,A -85,B 0,C 180,E1 14301.52,E2 14301.52} C_VEL
LIN {X 0,Y 309.278,Z 975.234,A -85,B 0,C 180,E1 14308.595,E2 14308.595} C_VEL
LIN {X 0,Y 308.85,Z 970.547,A -85,B 0,C 180,E1 14317.057,E2 14317.057} C_VEL
LIN {X 0,Y 309.967,Z 950.675,A -85,B 0,C 180,E1 14326.544,E2 14326.544} C_VEL
LIN {X 0,Y 314.857,Z 917.765,A -85,B 0,C 180,E1 14334.565,E2 14334.565} C_VEL
LIN {X 0,Y 322.399,Z 873.242,A -85,B 0,C 180,E1 14340.595,E2 14340.595} C_VEL
LIN {X 0,Y 328.67,Z 822.094,A -85,B 0,C 180,E1 14344.012,E2 14344.012} C_VEL
LIN {X 0,Y 313.769,Z 776.957,A -85,B 0,C 180,E1 14346.648,E2 14346.648} C_VEL
LIN {X 0,Y 299.04,Z 760.808,A -85,B 0,C 180,E1 14348.502,E2 14348.502} C_VEL
LIN {X 0,Y 296.989,Z 754.81,A -85,B 0,C 180,E1 14349.171,E2 14349.171} C_VEL
LIN {X 0,Y 296.8,Z 754.81,A -85,B 0,C 180,E1 14362.425,E2 14362.425} C_VEL
LIN {X 0,Y 297.261,Z 754.81,A -85,B 0,C 180,E1 14374.287,E2 14374.287} C_VEL
LIN {X 0,Y 298.177,Z 754.81,A -85,B 0,C 180,E1 14386.764,E2 14386.764} C_VEL
LIN {X 0,Y 299.006,Z 754.81,A -85,B 0,C 180,E1 14398.55,E2 14398.55} C_VEL
LIN {X 0,Y 298.489,Z 754.81,A -85,B 0,C 180,E1 14410.254,E2 14410.254} C_VEL
LIN {X 0,Y 297.61,Z 754.81,A -85,B 0,C 180,E1 14422.488,E2 14422.488} C_VEL
LIN {X 0,Y 296.935,Z 754.81,A -85,B 0,C 180,E1 14432.51,E2 14432.51} C_VEL
LIN {X 0,Y 296.722,Z 754.81,A -85,B 0,C 180,E1 14443.67,E2 14443.67} C_VEL
LIN {X 0,Y 296.778,Z 754.81,A -85,B 0,C 180,E1 14453.98,E2 14453.98} C_VEL
LIN {X 0,Y 297.129,Z 754.81,A -85,B 0,C 180,E1 14464.269,E2 14464.269} C_VEL
LIN {X 0,Y 297.954,Z 754.81,A -85,B 0,C 180,E1 14476.749,E2 14476.749} C_VEL
LIN {X 0,Y 298.506,Z 755.663,A -85,B 0,C 180,E1 14482.047,E2 14482.047} C_VEL
LIN {X 0,Y 311.025,Z 796.663,A -85,B 0,C 180,E1 14485.679,E2 14485.679} C_VEL
LIN {X 0,Y 312.732,Z 824.674,A -85,B 0,C 180,E1 14489.105,E2 14489.105} C_VEL
LIN {X 0,Y 306.762,Z 857.68,A -85,B 0,C 180,E1 14495.321,E2 14495.321} C_VEL
LIN {X 0,Y 302.963,Z 877.726,A -85,B 0,C 180,E1 14503.026,E2 14503.026} C_VEL
LIN {X 0,Y 302.237,Z 884.483,A -85,B 0,C 180,E1 14512.121,E2 14512.121} C_VEL
LIN {X 0,Y 305.493,Z 876.307,A -85,B 0,C 180,E1 14520.821,E2 14520.821} C_VEL
LIN {X 0,Y 312.476,Z 854.004,A -85,B 0,C 180,E1 14528.471,E2 14528.471} C_VEL
LIN {X 0,Y 320.235,Z 819.981,A -85,B 0,C 180,E1 14534.219,E2 14534.219} C_VEL
LIN {X 0,Y 310.141,Z 782.03,A -85,B 0,C 180,E1 14539.757,E2 14539.757} C_VEL
LIN {X 0,Y 297.001,Z 754.81,A -85,B 0,C 180,E1 14543.63,E2 14543.63} C_VEL
LIN {X 0,Y 297.193,Z 754.81,A -85,B 0,C 180,E1 14554.272,E2 14554.272} C_VEL
LIN {X 0,Y 297.936,Z 754.81,A -85,B 0,C 180,E1 14566.746,E2 14566.746} C_VEL
LIN {X 0,Y 299.304,Z 754.81,A -85,B 0,C 180,E1 14578.544,E2 14578.544} C_VEL
LIN {X 0,Y 298.355,Z 754.81,A -85,B 0,C 180,E1 14590.251,E2 14590.251} C_VEL
LIN {X 0,Y 297.59,Z 754.81,A -85,B 0,C 180,E1 14602.482,E2 14602.482} C_VEL
LIN {X 0,Y 297.049,Z 754.81,A -85,B 0,C 180,E1 14612.548,E2 14612.548} C_VEL
LIN {X 0,Y 296.86,Z 754.81,A -85,B 0,C 180,E1 14625.786,E2 14625.786} C_VEL
LIN {X 0,Y 321.445,Z 804.081,A -85,B 0,C 180,E1 14631.664,E2 14631.664} C_VEL
LIN {X 0,Y 327.111,Z 829.492,A -85,B 0,C 180,E1 14633.703,E2 14633.703} C_VEL
LIN {X 0,Y 318.335,Z 879.359,A -85,B 0,C 180,E1 14637.568,E2 14637.568} C_VEL
LIN {X 0,Y 308.395,Z 921.777,A -85,B 0,C 180,E1 14644.106,E2 14644.106} C_VEL
LIN {X 0,Y 301.954,Z 953.392,A -85,B 0,C 180,E1 14652.995,E2 14652.995} C_VEL
LIN {X 0,Y 300.801,Z 970.661,A -85,B 0,C 180,E1 14662.755,E2 14662.755} C_VEL
LIN {X 0,Y 301.324,Z 973.774,A -85,B 0,C 180,E1 14671.444,E2 14671.444} C_VEL
LIN {X 0,Y 300.799,Z 963.737,A -85,B 0,C 180,E1 14680.832,E2 14680.832} C_VEL
LIN {X 0,Y 303.164,Z 938.571,A -85,B 0,C 180,E1 14690.131,E2 14690.131} C_VEL
LIN {X 0,Y 310.023,Z 900.545,A -85,B 0,C 180,E1 14697.713,E2 14697.713} C_VEL
LIN {X 0,Y 318.031,Z 852.33,A -85,B 0,C 180,E1 14702.875,E2 14702.875} C_VEL
LIN {X 0,Y 319.871,Z 817.523,A -85,B 0,C 180,E1 14704.935,E2 14704.935} C_VEL
LIN {X 0,Y 299.04,Z 760.808,A -85,B 0,C 180,E1 14708.502,E2 14708.502} C_VEL
LIN {X 0,Y 293.193,Z 754.035,A -85,B 0,C 180,E1 14710.634,E2 14710.634} C_VEL
LIN {X 0,Y 288.77,Z 754.81,A -85,B 0,C 180,E1 14714.855,E2 14714.855} C_VEL
LIN {X 0,Y 288.84,Z 754.81,A -85,B 0,C 180,E1 14726.523,E2 14726.523} C_VEL
LIN {X 0,Y 289.637,Z 754.81,A -85,B 0,C 180,E1 14740.093,E2 14740.093} C_VEL
LIN {X 0,Y 290.666,Z 754.81,A -85,B 0,C 180,E1 14752.504,E2 14752.504} C_VEL
LIN {X 0,Y 290.784,Z 754.81,A -85,B 0,C 180,E1 14764.494,E2 14764.494} C_VEL
LIN {X 0,Y 289.935,Z 754.81,A -85,B 0,C 180,E1 14776.735,E2 14776.735} C_VEL
LIN {X 0,Y 288.993,Z 754.81,A -85,B 0,C 180,E1 14789.949,E2 14789.949} C_VEL
LIN {X 0,Y 288.682,Z 754.81,A -85,B 0,C 180,E1 14801.084,E2 14801.084} C_VEL
LIN {X 0,Y 288.726,Z 754.81,A -85,B 0,C 180,E1 14814.563,E2 14814.563} C_VEL
LIN {X 0,Y 289.185,Z 754.81,A -85,B 0,C 180,E1 14826.821,E2 14826.821} C_VEL
LIN {X 0,Y 290.191,Z 754.81,A -85,B 0,C 180,E1 14839.452,E2 14839.452} C_VEL
LIN {X 0,Y 290.531,Z 756.123,A -85,B 0,C 180,E1 14841.22,E2 14841.22} C_VEL
LIN {X 0,Y 303.512,Z 796.735,A -85,B 0,C 180,E1 14844.976,E2 14844.976} C_VEL
LIN {X 0,Y 305.106,Z 826.964,A -85,B 0,C 180,E1 14848.787,E2 14848.787} C_VEL
LIN {X 0,Y 298.882,Z 859.716,A -85,B 0,C 180,E1 14855.25,E2 14855.25} C_VEL
LIN {X 0,Y 294.914,Z 879.634,A -85,B 0,C 180,E1 14863.388,E2 14863.388} C_VEL
LIN {X 0,Y 294.459,Z 885.607,A -85,B 0,C 180,E1 14872.738,E2 14872.738} C_VEL
LIN {X 0,Y 298.243,Z 876.617,A -85,B 0,C 180,E1 14881.714,E2 14881.714} C_VEL
LIN {X 0,Y 305.942,Z 853.097,A -85,B 0,C 180,E1 14889.578,E2 14889.578} C_VEL
LIN {X 0,Y 312.995,Z 819.36,A -85,B 0,C 180,E1 14895.324,E2 14895.324} C_VEL
LIN {X 0,Y 302.279,Z 781.498,A -85,B 0,C 180,E1 14901.126,E2 14901.126} C_VEL
LIN {X 0,Y 288.846,Z 754.81,A -85,B 0,C 180,E1 14905.566,E2 14905.566} C_VEL
LIN {X 0,Y 289.213,Z 754.81,A -85,B 0,C 180,E1 14916.821,E2 14916.821} C_VEL
LIN {X 0,Y 290.172,Z 754.81,A -85,B 0,C 180,E1 14929.449,E2 14929.449} C_VEL
LIN {X 0,Y 290.989,Z 754.81,A -85,B 0,C 180,E1 14941.49,E2 14941.49} C_VEL
LIN {X 0,Y 289.97,Z 754.81,A -85,B 0,C 180,E1 14954.49,E2 14954.49} C_VEL
LIN {X 0,Y 289.278,Z 754.81,A -85,B 0,C 180,E1 14966.477,E2 14966.477} C_VEL
LIN {X 0,Y 288.879,Z 754.81,A -85,B 0,C 180,E1 14980.384,E2 14980.384} C_VEL
LIN {X 0,Y 289.027,Z 756.553,A -85,B 0,C 180,E1 14984.676,E2 14984.676} C_VEL
LIN {X 0,Y 315.237,Z 807.11,A -85,B 0,C 180,E1 14990.913,E2 14990.913} C_VEL
LIN {X 0,Y 320.299,Z 831.602,A -85,B 0,C 180,E1 14993,E2 14993} C_VEL
LIN {X 0,Y 310.863,Z 881.373,A -85,B 0,C 180,E1 14997.106,E2 14997.106} C_VEL
LIN {X 0,Y 300.599,Z 922.521,A -85,B 0,C 180,E1 15003.786,E2 15003.786} C_VEL
LIN {X 0,Y 293.982,Z 953.293,A -85,B 0,C 180,E1 15012.915,E2 15012.915} C_VEL
LIN {X 0,Y 292.85,Z 969.53,A -85,B 0,C 180,E1 15022.557,E2 15022.557} C_VEL
LIN {X 0,Y 293.425,Z 972.551,A -85,B 0,C 180,E1 15031.483,E2 15031.483} C_VEL
LIN {X 0,Y 292.898,Z 963.476,A -85,B 0,C 180,E1 15040.449,E2 15040.449} C_VEL
LIN {X 0,Y 295,Z 939.491,A -85,B 0,C 180,E1 15049.927,E2 15049.927} C_VEL
LIN {X 0,Y 302.073,Z 901.87,A -85,B 0,C 180,E1 15057.896,E2 15057.896} C_VEL
LIN {X 0,Y 310.353,Z 854.281,A -85,B 0,C 180,E1 15063.271,E2 15063.271} C_VEL
LIN {X 0,Y 312.335,Z 818.274,A -85,B 0,C 180,E1 15065.534,E2 15065.534} C_VEL
LIN {X 0,Y 288.948,Z 754.81,A -85,B 0,C 180,E1 15069.758,E2 15069.758} C_VEL
LIN {X 0,Y 288.77,Z 754.81,A -85,B 0,C 180,E1 15074.855,E2 15074.855} C_VEL
LIN {X 0,Y 280.668,Z 754.81,A -85,B 0,C 180,E1 15081.793,E2 15081.793} C_VEL
LIN {X 0,Y 281.099,Z 754.81,A -85,B 0,C 180,E1 15092.975,E2 15092.975} C_VEL
LIN {X 0,Y 282.047,Z 754.81,A -85,B 0,C 180,E1 15105.992,E2 15105.992} C_VEL
LIN {X 0,Y 282.989,Z 754.81,A -85,B 0,C 180,E1 15118.467,E2 15118.467} C_VEL
LIN {X 0,Y 282.376,Z 754.81,A -85,B 0,C 180,E1 15130.846,E2 15130.846} C_VEL
LIN {X 0,Y 281.359,Z 754.81,A -85,B 0,C 180,E1 15143.866,E2 15143.866} C_VEL
LIN {X 0,Y 280.73,Z 754.81,A -85,B 0,C 180,E1 15154.588,E2 15154.588} C_VEL
LIN {X 0,Y 280.528,Z 754.81,A -85,B 0,C 180,E1 15167.45,E2 15167.45} C_VEL
LIN {X 0,Y 280.8,Z 754.81,A -85,B 0,C 180,E1 15179.107,E2 15179.107} C_VEL
LIN {X 0,Y 281.511,Z 754.81,A -85,B 0,C 180,E1 15192.752,E2 15192.752} C_VEL
LIN {X 0,Y 282.34,Z 755.717,A -85,B 0,C 180,E1 15200.286,E2 15200.286} C_VEL
LIN {X 0,Y 296.208,Z 798.284,A -85,B 0,C 180,E1 15204.397,E2 15204.397} C_VEL
LIN {X 0,Y 297.557,Z 828.586,A -85,B 0,C 180,E1 15208.355,E2 15208.355} C_VEL
LIN {X 0,Y 291.098,Z 861.198,A -85,B 0,C 180,E1 15215.025,E2 15215.025} C_VEL
LIN {X 0,Y 286.9,Z 881.44,A -85,B 0,C 180,E1 15223.769,E2 15223.769} C_VEL
LIN {X 0,Y 286.672,Z 886.697,A -85,B 0,C 180,E1 15233.392,E2 15233.392} C_VEL
LIN {X 0,Y 290.809,Z 877.515,A -85,B 0,C 180,E1 15242.335,E2 15242.335} C_VEL
LIN {X 0,Y 298.815,Z 854.493,A -85,B 0,C 180,E1 15250.206,E2 15250.206} C_VEL
LIN {X 0,Y 306.198,Z 822.006,A -85,B 0,C 180,E1 15255.942,E2 15255.942} C_VEL
LIN {X 0,Y 296.135,Z 784.919,A -85,B 0,C 180,E1 15261.965,E2 15261.965} C_VEL
LIN {X 0,Y 280.852,Z 754.81,A -85,B 0,C 180,E1 15266.879,E2 15266.879} C_VEL
LIN {X 0,Y 281.312,Z 754.81,A -85,B 0,C 180,E1 15279.469,E2 15279.469} C_VEL
LIN {X 0,Y 282.453,Z 754.81,A -85,B 0,C 180,E1 15292.277,E2 15292.277} C_VEL
LIN {X 0,Y 282.975,Z 754.81,A -85,B 0,C 180,E1 15301.533,E2 15301.533} C_VEL
LIN {X 0,Y 282.032,Z 754.81,A -85,B 0,C 180,E1 15314.009,E2 15314.009} C_VEL
LIN {X 0,Y 281.151,Z 754.81,A -85,B 0,C 180,E1 15327.305,E2 15327.305} C_VEL
LIN {X 0,Y 280.798,Z 754.81,A -85,B 0,C 180,E1 15338.421,E2 15338.421} C_VEL
LIN {X 0,Y 280.915,Z 756.113,A -85,B 0,C 180,E1 15342.89,E2 15342.89} C_VEL
LIN {X 0,Y 307.621,Z 806.261,A -85,B 0,C 180,E1 15349.733,E2 15349.733} C_VEL
LIN {X 0,Y 313.731,Z 832.403,A -85,B 0,C 180,E1 15352.193,E2 15352.193} C_VEL
LIN {X 0,Y 303.722,Z 882.003,A -85,B 0,C 180,E1 15356.445,E2 15356.445} C_VEL
LIN {X 0,Y 292.827,Z 923.266,A -85,B 0,C 180,E1 15363.45,E2 15363.45} C_VEL
LIN {X 0,Y 285.905,Z 953.654,A -85,B 0,C 180,E1 15373.027,E2 15373.027} C_VEL
LIN {X 0,Y 284.882,Z 968.396,A -85,B 0,C 180,E1 15382.348,E2 15382.348} C_VEL
LIN {X 0,Y 285.498,Z 971.323,A -85,B 0,C 180,E1 15391.524,E2 15391.524} C_VEL
LIN {X 0,Y 284.906,Z 962.062,A -85,B 0,C 180,E1 15400.746,E2 15400.746} C_VEL
LIN {X 0,Y 287.323,Z 937.793,A -85,B 0,C 180,E1 15410.483,E2 15410.483} C_VEL
LIN {X 0,Y 294.564,Z 900.679,A -85,B 0,C 180,E1 15418.462,E2 15418.462} C_VEL
LIN {X 0,Y 303.006,Z 854.005,A -85,B 0,C 180,E1 15423.854,E2 15423.854} C_VEL
LIN {X 0,Y 305.02,Z 819.935,A -85,B 0,C 180,E1 15426.101,E2 15426.101} C_VEL
LIN {X 0,Y 280.869,Z 754.81,A -85,B 0,C 180,E1 15430.944,E2 15430.944} C_VEL
LIN {X 0,Y 280.668,Z 754.81,A -85,B 0,C 180,E1 15441.793,E2 15441.793} C_VEL
LIN {X 0,Y 272.816,Z 754.81,A -85,B 0,C 180,E1 15448.946,E2 15448.946} C_VEL
LIN {X 0,Y 273.708,Z 754.81,A -85,B 0,C 180,E1 15462.25,E2 15462.25} C_VEL
LIN {X 0,Y 274.767,Z 754.81,A -85,B 0,C 180,E1 15475.252,E2 15475.252} C_VEL
LIN {X 0,Y 274.74,Z 754.81,A -85,B 0,C 180,E1 15484.757,E2 15484.757} C_VEL
LIN {X 0,Y 273.787,Z 754.81,A -85,B 0,C 180,E1 15497.754,E2 15497.754} C_VEL
LIN {X 0,Y 272.838,Z 754.81,A -85,B 0,C 180,E1 15510.44,E2 15510.44} C_VEL
LIN {X 0,Y 272.417,Z 754.81,A -85,B 0,C 180,E1 15524.139,E2 15524.139} C_VEL
LIN {X 0,Y 272.767,Z 754.81,A -85,B 0,C 180,E1 15538.092,E2 15538.092} C_VEL
LIN {X 0,Y 273.441,Z 754.81,A -85,B 0,C 180,E1 15552.226,E2 15552.226} C_VEL
LIN {X 0,Y 274.176,Z 755.419,A -85,B 0,C 180,E1 15559.294,E2 15559.294} C_VEL
LIN {X 0,Y 288.82,Z 799.222,A -85,B 0,C 180,E1 15563.729,E2 15563.729} C_VEL
LIN {X 0,Y 290.053,Z 830.206,A -85,B 0,C 180,E1 15567.904,E2 15567.904} C_VEL
LIN {X 0,Y 283.43,Z 862.068,A -85,B 0,C 180,E1 15574.606,E2 15574.606} C_VEL
LIN {X 0,Y 279.069,Z 882.259,A -85,B 0,C 180,E1 15583.423,E2 15583.423} C_VEL
LIN {X 0,Y 278.337,Z 887.95,A -85,B 0,C 180,E1 15590.756,E2 15590.756} C_VEL
LIN {X 0,Y 281.761,Z 882.107,A -85,B 0,C 180,E1 15600.774,E2 15600.774} C_VEL
LIN {X 0,Y 289.793,Z 861.488,A -85,B 0,C 180,E1 15609.416,E2 15609.416} C_VEL
LIN {X 0,Y 299.607,Z 827.638,A -85,B 0,C 180,E1 15616.036,E2 15616.036} C_VEL
LIN {X 0,Y 291.388,Z 791.655,A -85,B 0,C 180,E1 15622.265,E2 15622.265} C_VEL
LIN {X 0,Y 272.859,Z 754.81,A -85,B 0,C 180,E1 15628.895,E2 15628.895} C_VEL
LIN {X 0,Y 273.438,Z 754.81,A -85,B 0,C 180,E1 15642.223,E2 15642.223} C_VEL
LIN {X 0,Y 274.694,Z 754.81,A -85,B 0,C 180,E1 15655.243,E2 15655.243} C_VEL
LIN {X 0,Y 274.733,Z 754.81,A -85,B 0,C 180,E1 15664.749,E2 15664.749} C_VEL
LIN {X 0,Y 273.725,Z 754.81,A -85,B 0,C 180,E1 15677.749,E2 15677.749} C_VEL
LIN {X 0,Y 272.892,Z 754.81,A -85,B 0,C 180,E1 15691.885,E2 15691.885} C_VEL
LIN {X 0,Y 272.84,Z 756.554,A -85,B 0,C 180,E1 15700.969,E2 15700.969} C_VEL
LIN {X 0,Y 299.328,Z 803.865,A -85,B 0,C 180,E1 15708.258,E2 15708.258} C_VEL
LIN {X 0,Y 307.203,Z 833.19,A -85,B 0,C 180,E1 15711.347,E2 15711.347} C_VEL
LIN {X 0,Y 296.978,Z 881.297,A -85,B 0,C 180,E1 15715.578,E2 15715.578} C_VEL
LIN {X 0,Y 285.528,Z 922.349,A -85,B 0,C 180,E1 15722.716,E2 15722.716} C_VEL
LIN {X 0,Y 278.105,Z 952.622,A -85,B 0,C 180,E1 15732.536,E2 15732.536} C_VEL
LIN {X 0,Y 276.938,Z 967.265,A -85,B 0,C 180,E1 15742.127,E2 15742.127} C_VEL
LIN {X 0,Y 277.577,Z 970.095,A -85,B 0,C 180,E1 15751.567,E2 15751.567} C_VEL
LIN {X 0,Y 276.919,Z 960.648,A -85,B 0,C 180,E1 15761.059,E2 15761.059} C_VEL
LIN {X 0,Y 279.588,Z 936.015,A -85,B 0,C 180,E1 15771.077,E2 15771.077} C_VEL
LIN {X 0,Y 287.36,Z 898.019,A -85,B 0,C 180,E1 15779.284,E2 15779.284} C_VEL
LIN {X 0,Y 296.088,Z 851.119,A -85,B 0,C 180,E1 15784.674,E2 15784.674} C_VEL
LIN {X 0,Y 297.77,Z 821.813,A -85,B 0,C 180,E1 15786.68,E2 15786.68} C_VEL
LIN {X 0,Y 272.726,Z 754.81,A -85,B 0,C 180,E1 15792.067,E2 15792.067} C_VEL
LIN {X 0,Y 272.616,Z 754.81,A -85,B 0,C 180,E1 15804.238,E2 15804.238} C_VEL
LIN {X 0,Y 272.816,Z 754.81,A -85,B 0,C 180,E1 15808.946,E2 15808.946} C_VEL
LIN {X 0,Y 265.036,Z 754.81,A -85,B 0,C 180,E1 15816.363,E2 15816.363} C_VEL
LIN {X 0,Y 266.19,Z 754.81,A -85,B 0,C 180,E1 15828.494,E2 15828.494} C_VEL
LIN {X 0,Y 267.234,Z 754.81,A -85,B 0,C 180,E1 15841.631,E2 15841.631} C_VEL
LIN {X 0,Y 265.962,Z 754.81,A -85,B 0,C 180,E1 15854.882,E2 15854.882} C_VEL
LIN {X 0,Y 264.917,Z 754.81,A -85,B 0,C 180,E1 15867.385,E2 15867.385} C_VEL
LIN {X 0,Y 264.432,Z 754.81,A -85,B 0,C 180,E1 15881.303,E2 15881.303} C_VEL
LIN {X 0,Y 264.44,Z 754.81,A -85,B 0,C 180,E1 15892.944,E2 15892.944} C_VEL
LIN {X 0,Y 264.868,Z 754.81,A -85,B 0,C 180,E1 15904.549,E2 15904.549} C_VEL
LIN {X 0,Y 266.164,Z 756.598,A -85,B 0,C 180,E1 15918.317,E2 15918.317} C_VEL
LIN {X 0,Y 281.239,Z 798.407,A -85,B 0,C 180,E1 15922.824,E2 15922.824} C_VEL
LIN {X 0,Y 282.663,Z 830.95,A -85,B 0,C 180,E1 15927.306,E2 15927.306} C_VEL
LIN {X 0,Y 275.657,Z 863.47,A -85,B 0,C 180,E1 15934.34,E2 15934.34} C_VEL
LIN {X 0,Y 271.205,Z 883.22,A -85,B 0,C 180,E1 15943.187,E2 15943.187} C_VEL
LIN {X 0,Y 270.628,Z 889.282,A -85,B 0,C 180,E1 15952.285,E2 15952.285} C_VEL
LIN {X 0,Y 274.481,Z 882.696,A -85,B 0,C 180,E1 15961.683,E2 15961.683} C_VEL
LIN {X 0,Y 283.187,Z 861.255,A -85,B 0,C 180,E1 15970.523,E2 15970.523} C_VEL
LIN {X 0,Y 292.671,Z 827.768,A -85,B 0,C 180,E1 15977.157,E2 15977.157} C_VEL
LIN {X 0,Y 284.39,Z 792.579,A -85,B 0,C 180,E1 15983.579,E2 15983.579} C_VEL
LIN {X 0,Y 264.85,Z 754.81,A -85,B 0,C 180,E1 15991.336,E2 15991.336} C_VEL
LIN {X 0,Y 265.638,Z 754.81,A -85,B 0,C 180,E1 16005.099,E2 16005.099} C_VEL
LIN {X 0,Y 267.217,Z 754.81,A -85,B 0,C 180,E1 16018.369,E2 16018.369} C_VEL
LIN {X 0,Y 266.13,Z 754.81,A -85,B 0,C 180,E1 16031.508,E2 16031.508} C_VEL
LIN {X 0,Y 265.09,Z 754.81,A -85,B 0,C 180,E1 16045.422,E2 16045.422} C_VEL
LIN {X 0,Y 264.659,Z 756.064,A -85,B 0,C 180,E1 16058.727,E2 16058.727} C_VEL
LIN {X 0,Y 291.197,Z 801.979,A -85,B 0,C 180,E1 16066.711,E2 16066.711} C_VEL
LIN {X 0,Y 300.704,Z 834.424,A -85,B 0,C 180,E1 16070.496,E2 16070.496} C_VEL
LIN {X 0,Y 289.947,Z 882.009,A -85,B 0,C 180,E1 16074.85,E2 16074.85} C_VEL
LIN {X 0,Y 277.769,Z 923.059,A -85,B 0,C 180,E1 16082.33,E2 16082.33} C_VEL
LIN {X 0,Y 270.068,Z 952.732,A -85,B 0,C 180,E1 16092.577,E2 16092.577} C_VEL
LIN {X 0,Y 269.118,Z 967.423,A -85,B 0,C 180,E1 16103.525,E2 16103.525} C_VEL
LIN {X 0,Y 269.647,Z 968.863,A -85,B 0,C 180,E1 16111.614,E2 16111.614} C_VEL
LIN {X 0,Y 268.933,Z 959.202,A -85,B 0,C 180,E1 16121.392,E2 16121.392} C_VEL
LIN {X 0,Y 271.842,Z 934.527,A -85,B 0,C 180,E1 16131.602,E2 16131.602} C_VEL
LIN {X 0,Y 279.8,Z 897.444,A -85,B 0,C 180,E1 16139.815,E2 16139.815} C_VEL
LIN {X 0,Y 288.79,Z 850.905,A -85,B 0,C 180,E1 16145.318,E2 16145.318} C_VEL
LIN {X 0,Y 290.169,Z 822.489,A -85,B 0,C 180,E1 16147.367,E2 16147.367} C_VEL
LIN {X 0,Y 264.685,Z 754.81,A -85,B 0,C 180,E1 16152.807,E2 16152.807} C_VEL
LIN {X 0,Y 264.634,Z 754.81,A -85,B 0,C 180,E1 16166.995,E2 16166.995} C_VEL
LIN {X 0,Y 265.036,Z 754.81,A -85,B 0,C 180,E1 16176.363,E2 16176.363} C_VEL
LIN {X 0,Y 257.667,Z 754.81,A -85,B 0,C 180,E1 16184.027,E2 16184.027} C_VEL
LIN {X 0,Y 258.752,Z 754.81,A -85,B 0,C 180,E1 16194.957,E2 16194.957} C_VEL
LIN {X 0,Y 258.698,Z 754.81,A -85,B 0,C 180,E1 16205.052,E2 16205.052} C_VEL
LIN {X 0,Y 257.592,Z 754.81,A -85,B 0,C 180,E1 16218.911,E2 16218.911} C_VEL
LIN {X 0,Y 256.608,Z 754.81,A -85,B 0,C 180,E1 16230.958,E2 16230.958} C_VEL
LIN {X 0,Y 256.347,Z 754.81,A -85,B 0,C 180,E1 16242.911,E2 16242.911} C_VEL
LIN {X 0,Y 256.471,Z 754.81,A -85,B 0,C 180,E1 16255.796,E2 16255.796} C_VEL
LIN {X 0,Y 256.978,Z 754.81,A -85,B 0,C 180,E1 16267.426,E2 16267.426} C_VEL
LIN {X 0,Y 258.089,Z 756.718,A -85,B 0,C 180,E1 16277.228,E2 16277.228} C_VEL
LIN {X 0,Y 273.709,Z 799.137,A -85,B 0,C 180,E1 16282.031,E2 16282.031} C_VEL
LIN {X 0,Y 275.155,Z 832.655,A -85,B 0,C 180,E1 16286.837,E2 16286.837} C_VEL
LIN {X 0,Y 267.892,Z 864.849,A -85,B 0,C 180,E1 16294.06,E2 16294.06} C_VEL
LIN {X 0,Y 263.239,Z 884.672,A -85,B 0,C 180,E1 16303.331,E2 16303.331} C_VEL
LIN {X 0,Y 262.693,Z 890.48,A -85,B 0,C 180,E1 16312.054,E2 16312.054} C_VEL
LIN {X 0,Y 266.408,Z 884.831,A -85,B 0,C 180,E1 16321.499,E2 16321.499} C_VEL
LIN {X 0,Y 275.403,Z 864.495,A -85,B 0,C 180,E1 16330.688,E2 16330.688} C_VEL
LIN {X 0,Y 286.005,Z 831.67,A -85,B 0,C 180,E1 16337.598,E2 16337.598} C_VEL
LIN {X 0,Y 278.547,Z 796.453,A -85,B 0,C 180,E1 16344.437,E2 16344.437} C_VEL
LIN {X 0,Y 259.386,Z 760.632,A -85,B 0,C 180,E1 16352.257,E2 16352.257} C_VEL
LIN {X 0,Y 256.871,Z 754.81,A -85,B 0,C 180,E1 16353.694,E2 16353.694} C_VEL
LIN {X 0,Y 257.897,Z 754.81,A -85,B 0,C 180,E1 16368.11,E2 16368.11} C_VEL
LIN {X 0,Y 259.205,Z 754.81,A -85,B 0,C 180,E1 16378.318,E2 16378.318} C_VEL
LIN {X 0,Y 258.05,Z 754.81,A -85,B 0,C 180,E1 16391.874,E2 16391.874} C_VEL
LIN {X 0,Y 257.088,Z 754.81,A -85,B 0,C 180,E1 16403.803,E2 16403.803} C_VEL
LIN {X 0,Y 256.663,Z 756.032,A -85,B 0,C 180,E1 16416.284,E2 16416.284} C_VEL
LIN {X 0,Y 282.737,Z 799.53,A -85,B 0,C 180,E1 16424.916,E2 16424.916} C_VEL
LIN {X 0,Y 294.219,Z 835.933,A -85,B 0,C 180,E1 16429.613,E2 16429.613} C_VEL
LIN {X 0,Y 282.45,Z 884.442,A -85,B 0,C 180,E1 16434.343,E2 16434.343} C_VEL
LIN {X 0,Y 270.036,Z 923.715,A -85,B 0,C 180,E1 16441.924,E2 16441.924} C_VEL
LIN {X 0,Y 262.144,Z 952.342,A -85,B 0,C 180,E1 16452.368,E2 16452.368} C_VEL
LIN {X 0,Y 261.141,Z 966.281,A -85,B 0,C 180,E1 16463.327,E2 16463.327} C_VEL
LIN {X 0,Y 261.724,Z 967.628,A -85,B 0,C 180,E1 16471.662,E2 16471.662} C_VEL
LIN {X 0,Y 260.98,Z 957.727,A -85,B 0,C 180,E1 16481.744,E2 16481.744} C_VEL
LIN {X 0,Y 264.002,Z 933.753,A -85,B 0,C 180,E1 16491.942,E2 16491.942} C_VEL
LIN {X 0,Y 272.271,Z 896.865,A -85,B 0,C 180,E1 16500.37,E2 16500.37} C_VEL
LIN {X 0,Y 281.758,Z 849.178,A -85,B 0,C 180,E1 16506.103,E2 16506.103} C_VEL
LIN {X 0,Y 282.76,Z 823.838,A -85,B 0,C 180,E1 16508.02,E2 16508.02} C_VEL
LIN {X 0,Y 258.833,Z 760.846,A -85,B 0,C 180,E1 16513.321,E2 16513.321} C_VEL
LIN {X 0,Y 256.546,Z 754.81,A -85,B 0,C 180,E1 16514.059,E2 16514.059} C_VEL
LIN {X 0,Y 256.534,Z 754.81,A -85,B 0,C 180,E1 16525.812,E2 16525.812} C_VEL
LIN {X 0,Y 257.172,Z 754.81,A -85,B 0,C 180,E1 16537.45,E2 16537.45} C_VEL
LIN {X 0,Y 257.667,Z 754.81,A -85,B 0,C 180,E1 16544.027,E2 16544.027} C_VEL
LIN {X 0,Y 250.379,Z 754.81,A -85,B 0,C 180,E1 16551.889,E2 16551.889} C_VEL
LIN {X 0,Y 250.843,Z 754.81,A -85,B 0,C 180,E1 16563.386,E2 16563.386} C_VEL
LIN {X 0,Y 249.763,Z 754.81,A -85,B 0,C 180,E1 16575.872,E2 16575.872} C_VEL
LIN {X 0,Y 248.727,Z 754.81,A -85,B 0,C 180,E1 16587.783,E2 16587.783} C_VEL
LIN {X 0,Y 248.225,Z 754.81,A -85,B 0,C 180,E1 16600.161,E2 16600.161} C_VEL
LIN {X 0,Y 248.451,Z 754.81,A -85,B 0,C 180,E1 16615.554,E2 16615.554} C_VEL
LIN {X 0,Y 249.154,Z 754.81,A -85,B 0,C 180,E1 16630.426,E2 16630.426} C_VEL
LIN {X 0,Y 249.764,Z 755.835,A -85,B 0,C 180,E1 16635.979,E2 16635.979} C_VEL
LIN {X 0,Y 265.88,Z 798.465,A -85,B 0,C 180,E1 16641.005,E2 16641.005} C_VEL
LIN {X 0,Y 267.851,Z 833.234,A -85,B 0,C 180,E1 16646.149,E2 16646.149} C_VEL
LIN {X 0,Y 260.141,Z 866.225,A -85,B 0,C 180,E1 16653.762,E2 16653.762} C_VEL
LIN {X 0,Y 255.458,Z 885.367,A -85,B 0,C 180,E1 16662.871,E2 16662.871} C_VEL
LIN {X 0,Y 254.91,Z 891.671,A -85,B 0,C 180,E1 16672.765,E2 16672.765} C_VEL
LIN {X 0,Y 259.248,Z 885.385,A -85,B 0,C 180,E1 16682.545,E2 16682.545} C_VEL
LIN {X 0,Y 268.822,Z 864.753,A -85,B 0,C 180,E1 16691.773,E2 16691.773} C_VEL
LIN {X 0,Y 279.216,Z 831.887,A -85,B 0,C 180,E1 16698.822,E2 16698.822} C_VEL
LIN {X 0,Y 271.623,Z 797.126,A -85,B 0,C 180,E1 16705.956,E2 16705.956} C_VEL
LIN {X 0,Y 252.399,Z 761.473,A -85,B 0,C 180,E1 16714.523,E2 16714.523} C_VEL
LIN {X 0,Y 248.93,Z 754.81,A -85,B 0,C 180,E1 16716.651,E2 16716.651} C_VEL
LIN {X 0,Y 250.214,Z 754.81,A -85,B 0,C 180,E1 16731.274,E2 16731.274} C_VEL
LIN {X 0,Y 250.747,Z 754.81,A -85,B 0,C 180,E1 16743.034,E2 16743.034} C_VEL
LIN {X 0,Y 249.682,Z 754.81,A -85,B 0,C 180,E1 16755.868,E2 16755.868} C_VEL
LIN {X 0,Y 248.777,Z 754.81,A -85,B 0,C 180,E1 16767.81,E2 16767.81} C_VEL
LIN {X 0,Y 248.834,Z 756.735,A -85,B 0,C 180,E1 16773.547,E2 16773.547} C_VEL
LIN {X 0,Y 273.197,Z 795.199,A -85,B 0,C 180,E1 16782.603,E2 16782.603} C_VEL
LIN {X 0,Y 287.763,Z 834.76,A -85,B 0,C 180,E1 16788.428,E2 16788.428} C_VEL
LIN {X 0,Y 275.988,Z 883.514,A -85,B 0,C 180,E1 16793.317,E2 16793.317} C_VEL
LIN {X 0,Y 262.843,Z 922.851,A -85,B 0,C 180,E1 16801.084,E2 16801.084} C_VEL
LIN {X 0,Y 254.395,Z 951.051,A -85,B 0,C 180,E1 16811.655,E2 16811.655} C_VEL
LIN {X 0,Y 253.045,Z 964.144,A -85,B 0,C 180,E1 16821.671,E2 16821.671} C_VEL
LIN {X 0,Y 253.79,Z 966.391,A -85,B 0,C 180,E1 16831.714,E2 16831.714} C_VEL
LIN {X 0,Y 253.046,Z 956.245,A -85,B 0,C 180,E1 16842.118,E2 16842.118} C_VEL
LIN {X 0,Y 256.384,Z 931.9,A -85,B 0,C 180,E1 16852.629,E2 16852.629} C_VEL
LIN {X 0,Y 265.087,Z 894.608,A -85,B 0,C 180,E1 16861.226,E2 16861.226} C_VEL
LIN {X 0,Y 274.739,Z 847.61,A -85,B 0,C 180,E1 16866.915,E2 16866.915} C_VEL
LIN {X 0,Y 275.322,Z 825.092,A -85,B 0,C 180,E1 16868.721,E2 16868.721} C_VEL
LIN {X 0,Y 253.655,Z 767.081,A -85,B 0,C 180,E1 16873.863,E2 16873.863} C_VEL
LIN {X 0,Y 248.425,Z 754.81,A -85,B 0,C 180,E1 16875.379,E2 16875.379} C_VEL
LIN {X 0,Y 248.589,Z 754.81,A -85,B 0,C 180,E1 16888.747,E2 16888.747} C_VEL
LIN {X 0,Y 249.404,Z 754.81,A -85,B 0,C 180,E1 16900.59,E2 16900.59} C_VEL
LIN {X 0,Y 250.379,Z 754.81,A -85,B 0,C 180,E1 16911.889,E2 16911.889} C_VEL
LIN {X 0,Y 242.943,Z 754.81,A -85,B 0,C 180,E1 16919.977,E2 16919.977} C_VEL
LIN {X 0,Y 241.878,Z 754.81,A -85,B 0,C 180,E1 16933.465,E2 16933.465} C_VEL
LIN {X 0,Y 240.667,Z 754.81,A -85,B 0,C 180,E1 16948.229,E2 16948.229} C_VEL
LIN {X 0,Y 240.06,Z 754.81,A -85,B 0,C 180,E1 16963.364,E2 16963.364} C_VEL
LIN {X 0,Y 240.49,Z 754.81,A -85,B 0,C 180,E1 16978.426,E2 16978.426} C_VEL
LIN {X 0,Y 241.356,Z 754.81,A -85,B 0,C 180,E1 16993.563,E2 16993.563} C_VEL
LIN {X 0,Y 241.833,Z 756.975,A -85,B 0,C 180,E1 16994.783,E2 16994.783} C_VEL
LIN {X 0,Y 258.013,Z 797.969,A -85,B 0,C 180,E1 16999.948,E2 16999.948} C_VEL
LIN {X 0,Y 260.748,Z 832.999,A -85,B 0,C 180,E1 17005.295,E2 17005.295} C_VEL
LIN {X 0,Y 252.712,Z 866.04,A -85,B 0,C 180,E1 17012.905,E2 17012.905} C_VEL
LIN {X 0,Y 247.655,Z 886.002,A -85,B 0,C 180,E1 17022.383,E2 17022.383} C_VEL
LIN {X 0,Y 247.18,Z 892.866,A -85,B 0,C 180,E1 17033.519,E2 17033.519} C_VEL
LIN {X 0,Y 252.182,Z 885.779,A -85,B 0,C 180,E1 17043.716,E2 17043.716} C_VEL
LIN {X 0,Y 262.556,Z 864.468,A -85,B 0,C 180,E1 17053.05,E2 17053.05} C_VEL
LIN {X 0,Y 272.53,Z 833.502,A -85,B 0,C 180,E1 17059.82,E2 17059.82} C_VEL
LIN {X 0,Y 265.528,Z 800.058,A -85,B 0,C 180,E1 17067.111,E2 17067.111} C_VEL
LIN {X 0,Y 248.371,Z 767.432,A -85,B 0,C 180,E1 17075.638,E2 17075.638} C_VEL
LIN {X 0,Y 241.037,Z 754.81,A -85,B 0,C 180,E1 17079.735,E2 17079.735} C_VEL
LIN {X 0,Y 242.568,Z 754.81,A -85,B 0,C 180,E1 17094.611,E2 17094.611} C_VEL
LIN {X 0,Y 242.612,Z 754.81,A -85,B 0,C 180,E1 17105.379,E2 17105.379} C_VEL
LIN {X 0,Y 241.279,Z 754.81,A -85,B 0,C 180,E1 17120.234,E2 17120.234} C_VEL
LIN {X 0,Y 240.775,Z 756.438,A -85,B 0,C 180,E1 17130.183,E2 17130.183} C_VEL
LIN {X 0,Y 264.576,Z 792.844,A -85,B 0,C 180,E1 17140.315,E2 17140.315} C_VEL
LIN {X 0,Y 280.086,Z 831.369,A -85,B 0,C 180,E1 17146.727,E2 17146.727} C_VEL
LIN {X 0,Y 279.619,Z 847.033,A -85,B 0,C 180,E1 17148.359,E2 17148.359} C_VEL
LIN {X 0,Y 266.362,Z 892.439,A -85,B 0,C 180,E1 17153.766,E2 17153.766} C_VEL
LIN {X 0,Y 253.08,Z 929.125,A -85,B 0,C 180,E1 17162.309,E2 17162.309} C_VEL
LIN {X 0,Y 245.499,Z 954.645,A -85,B 0,C 180,E1 17173.85,E2 17173.85} C_VEL
LIN {X 0,Y 245.415,Z 964.899,A -85,B 0,C 180,E1 17184.679,E2 17184.679} C_VEL
LIN {X 0,Y 245.588,Z 963.128,A -85,B 0,C 180,E1 17195.32,E2 17195.32} C_VEL
LIN {X 0,Y 246.238,Z 946.079,A -85,B 0,C 180,E1 17207.22,E2 17207.22} C_VEL
LIN {X 0,Y 252.831,Z 914.147,A -85,B 0,C 180,E1 17217.723,E2 17217.723} C_VEL
LIN {X 0,Y 262.92,Z 870.782,A -85,B 0,C 180,E1 17225.255,E2 17225.255} C_VEL
LIN {X 0,Y 268.558,Z 828.696,A -85,B 0,C 180,E1 17229.214,E2 17229.214} C_VEL
LIN {X 0,Y 248.856,Z 773.666,A -85,B 0,C 180,E1 17234.361,E2 17234.361} C_VEL
LIN {X 0,Y 240.246,Z 754.81,A -85,B 0,C 180,E1 17236.589,E2 17236.589} C_VEL
LIN {X 0,Y 240.65,Z 754.81,A -85,B 0,C 180,E1 17251.779,E2 17251.779} C_VEL
LIN {X 0,Y 241.834,Z 754.81,A -85,B 0,C 180,E1 17266.579,E2 17266.579} C_VEL
LIN {X 0,Y 242.943,Z 754.81,A -85,B 0,C 180,E1 17279.977,E2 17279.977} C_VEL
LIN {X 0,Y 234.217,Z 754.81,A -85,B 0,C 180,E1 17288.298,E2 17288.298} C_VEL
LIN {X 0,Y 233.166,Z 754.81,A -85,B 0,C 180,E1 17300.98,E2 17300.98} C_VEL
LIN {X 0,Y 232.107,Z 754.81,A -85,B 0,C 180,E1 17315.184,E2 17315.184} C_VEL
LIN {X 0,Y 232.029,Z 754.81,A -85,B 0,C 180,E1 17328.783,E2 17328.783} C_VEL
LIN {X 0,Y 232.574,Z 754.81,A -85,B 0,C 180,E1 17341.758,E2 17341.758} C_VEL
LIN {X 0,Y 233.454,Z 756.277,A -85,B 0,C 180,E1 17353.345,E2 17353.345} C_VEL
LIN {X 0,Y 250.472,Z 798.592,A -85,B 0,C 180,E1 17358.976,E2 17358.976} C_VEL
LIN {X 0,Y 253.831,Z 831.934,A -85,B 0,C 180,E1 17364.275,E2 17364.275} C_VEL
LIN {X 0,Y 245.51,Z 865.013,A -85,B 0,C 180,E1 17371.77,E2 17371.77} C_VEL
LIN {X 0,Y 240.023,Z 886.073,A -85,B 0,C 180,E1 17381.458,E2 17381.458} C_VEL
LIN {X 0,Y 239.158,Z 894.069,A -85,B 0,C 180,E1 17393.05,E2 17393.05} C_VEL
LIN {X 0,Y 244.556,Z 887.281,A -85,B 0,C 180,E1 17404.146,E2 17404.146} C_VEL
LIN {X 0,Y 255.414,Z 866.43,A -85,B 0,C 180,E1 17413.73,E2 17413.73} C_VEL
LIN {X 0,Y 265.922,Z 835.801,A -85,B 0,C 180,E1 17420.727,E2 17420.727} C_VEL
LIN {X 0,Y 259.674,Z 803.237,A -85,B 0,C 180,E1 17428.26,E2 17428.26} C_VEL
LIN {X 0,Y 243.653,Z 771.859,A -85,B 0,C 180,E1 17437.16,E2 17437.16} C_VEL
LIN {X 0,Y 233.363,Z 754.81,A -85,B 0,C 180,E1 17443.951,E2 17443.951} C_VEL
LIN {X 0,Y 235.128,Z 754.81,A -85,B 0,C 180,E1 17458.146,E2 17458.146} C_VEL
LIN {X 0,Y 234.172,Z 754.81,A -85,B 0,C 180,E1 17469.319,E2 17469.319} C_VEL
LIN {X 0,Y 233.143,Z 754.81,A -85,B 0,C 180,E1 17480.972,E2 17480.972} C_VEL
LIN {X 0,Y 232.943,Z 756.732,A -85,B 0,C 180,E1 17486.198,E2 17486.198} C_VEL
LIN {X 0,Y 252.849,Z 785.585,A -85,B 0,C 180,E1 17496.471,E2 17496.471} C_VEL
LIN {X 0,Y 271.054,Z 823.473,A -85,B 0,C 180,E1 17504.109,E2 17504.109} C_VEL
LIN {X 0,Y 274.355,Z 843.899,A -85,B 0,C 180,E1 17507.023,E2 17507.023} C_VEL
LIN {X 0,Y 260.263,Z 890.62,A -85,B 0,C 180,E1 17512.513,E2 17512.513} C_VEL
LIN {X 0,Y 245.854,Z 928.29,A -85,B 0,C 180,E1 17521.422,E2 17521.422} C_VEL
LIN {X 0,Y 237.701,Z 953.605,A -85,B 0,C 180,E1 17533.305,E2 17533.305} C_VEL
LIN {X 0,Y 237.45,Z 963.742,A -85,B 0,C 180,E1 17544.5,E2 17544.5} C_VEL
LIN {X 0,Y 237.645,Z 961.808,A -85,B 0,C 180,E1 17555.498,E2 17555.498} C_VEL
LIN {X 0,Y 238.355,Z 944.429,A -85,B 0,C 180,E1 17567.808,E2 17567.808} C_VEL
LIN {X 0,Y 245.074,Z 913.828,A -85,B 0,C 180,E1 17578.176,E2 17578.176} C_VEL
LIN {X 0,Y 255.364,Z 871.561,A -85,B 0,C 180,E1 17585.833,E2 17585.833} C_VEL
LIN {X 0,Y 261.551,Z 831.481,A -85,B 0,C 180,E1 17589.78,E2 17589.78} C_VEL
LIN {X 0,Y 243.471,Z 779.108,A -85,B 0,C 180,E1 17595.003,E2 17595.003} C_VEL
LIN {X 0,Y 232.203,Z 754.81,A -85,B 0,C 180,E1 17597.789,E2 17597.789} C_VEL
LIN {X 0,Y 232.658,Z 754.81,A -85,B 0,C 180,E1 17611.714,E2 17611.714} C_VEL
LIN {X 0,Y 233.868,Z 754.81,A -85,B 0,C 180,E1 17626.878,E2 17626.878} C_VEL
LIN {X 0,Y 234.924,Z 754.81,A -85,B 0,C 180,E1 17640.001,E2 17640.001} C_VEL
LIN {X 0,Y 234.217,Z 754.81,A -85,B 0,C 180,E1 17648.298,E2 17648.298} C_VEL
LIN {X 0,Y 225.424,Z 754.81,A -85,B 0,C 180,E1 17656.939,E2 17656.939} C_VEL
LIN {X 0,Y 224.182,Z 754.81,A -85,B 0,C 180,E1 17672.2,E2 17672.2} C_VEL
LIN {X 0,Y 223.991,Z 754.81,A -85,B 0,C 180,E1 17685.354,E2 17685.354} C_VEL
LIN {X 0,Y 224.252,Z 754.81,A -85,B 0,C 180,E1 17699.498,E2 17699.498} C_VEL
LIN {X 0,Y 225.273,Z 756.534,A -85,B 0,C 180,E1 17711.849,E2 17711.849} C_VEL
LIN {X 0,Y 242.908,Z 798.763,A -85,B 0,C 180,E1 17717.881,E2 17717.881} C_VEL
LIN {X 0,Y 246.614,Z 832.725,A -85,B 0,C 180,E1 17723.511,E2 17723.511} C_VEL
LIN {X 0,Y 237.798,Z 866.376,A -85,B 0,C 180,E1 17731.37,E2 17731.37} C_VEL
LIN {X 0,Y 231.932,Z 887.943,A -85,B 0,C 180,E1 17741.863,E2 17741.863} C_VEL
LIN {X 0,Y 230.933,Z 894.984,A -85,B 0,C 180,E1 17751.187,E2 17751.187} C_VEL
LIN {X 0,Y 235.805,Z 890.441,A -85,B 0,C 180,E1 17763.162,E2 17763.162} C_VEL
LIN {X 0,Y 246.955,Z 871.139,A -85,B 0,C 180,E1 17773.521,E2 17773.521} C_VEL
LIN {X 0,Y 259.429,Z 840.107,A -85,B 0,C 180,E1 17781.18,E2 17781.18} C_VEL
LIN {X 0,Y 254.405,Z 808.139,A -85,B 0,C 180,E1 17789.031,E2 17789.031} C_VEL
LIN {X 0,Y 238.991,Z 775.588,A -85,B 0,C 180,E1 17798.881,E2 17798.881} C_VEL
LIN {X 0,Y 227.044,Z 759.307,A -85,B 0,C 180,E1 17807.02,E2 17807.02} C_VEL
LIN {X 0,Y 225.764,Z 754.81,A -85,B 0,C 180,E1 17808.915,E2 17808.915} C_VEL
LIN {X 0,Y 226.89,Z 754.81,A -85,B 0,C 180,E1 17821.912,E2 17821.912} C_VEL
LIN {X 0,Y 225.739,Z 754.81,A -85,B 0,C 180,E1 17833.604,E2 17833.604} C_VEL
LIN {X 0,Y 225.391,Z 756.903,A -85,B 0,C 180,E1 17841.118,E2 17841.118} C_VEL
LIN {X 0,Y 241.074,Z 779.01,A -85,B 0,C 180,E1 17851.72,E2 17851.72} C_VEL
LIN {X 0,Y 260.056,Z 812.835,A -85,B 0,C 180,E1 17860.475,E2 17860.475} C_VEL
LIN {X 0,Y 268.301,Z 844.643,A -85,B 0,C 180,E1 17865.932,E2 17865.932} C_VEL
LIN {X 0,Y 253.881,Z 890.009,A -85,B 0,C 180,E1 17871.4,E2 17871.4} C_VEL
LIN {X 0,Y 238.7,Z 927.444,A -85,B 0,C 180,E1 17880.482,E2 17880.482} C_VEL
LIN {X 0,Y 229.911,Z 952.569,A -85,B 0,C 180,E1 17892.722,E2 17892.722} C_VEL
LIN {X 0,Y 229.478,Z 962.583,A -85,B 0,C 180,E1 17904.308,E2 17904.308} C_VEL
LIN {X 0,Y 229.714,Z 960.488,A -85,B 0,C 180,E1 17915.688,E2 17915.688} C_VEL
LIN {X 0,Y 230.463,Z 943.185,A -85,B 0,C 180,E1 17928.228,E2 17928.228} C_VEL
LIN {X 0,Y 237.701,Z 911.956,A -85,B 0,C 180,E1 17939.04,E2 17939.04} C_VEL
LIN {X 0,Y 248.561,Z 869.082,A -85,B 0,C 180,E1 17946.849,E2 17946.849} C_VEL
LIN {X 0,Y 254.334,Z 833.37,A -85,B 0,C 180,E1 17950.475,E2 17950.475} C_VEL
LIN {X 0,Y 237.47,Z 783.079,A -85,B 0,C 180,E1 17955.823,E2 17955.823} C_VEL
LIN {X 0,Y 224.107,Z 754.81,A -85,B 0,C 180,E1 17959.594,E2 17959.594} C_VEL
LIN {X 0,Y 224.676,Z 754.81,A -85,B 0,C 180,E1 17973.963,E2 17973.963} C_VEL
LIN {X 0,Y 225.876,Z 754.81,A -85,B 0,C 180,E1 17986.963,E2 17986.963} C_VEL
LIN {X 0,Y 226.926,Z 754.81,A -85,B 0,C 180,E1 17998.089,E2 17998.089} C_VEL
LIN {X 0,Y 226.14,Z 754.81,A -85,B 0,C 180,E1 18009.663,E2 18009.663} C_VEL
LIN {X 0,Y 225.424,Z 754.81,A -85,B 0,C 180,E1 18016.939,E2 18016.939} C_VEL
LIN {X 0,Y 216.452,Z 754.81,A -85,B 0,C 180,E1 18025.921,E2 18025.921} C_VEL
LIN {X 0,Y 215.804,Z 754.81,A -85,B 0,C 180,E1 18041.923,E2 18041.923} C_VEL
LIN {X 0,Y 216.166,Z 754.81,A -85,B 0,C 180,E1 18058.227,E2 18058.227} C_VEL
LIN {X 0,Y 217.093,Z 756.398,A -85,B 0,C 180,E1 18070.209,E2 18070.209} C_VEL
LIN {X 0,Y 234.953,Z 797.621,A -85,B 0,C 180,E1 18076.51,E2 18076.51} C_VEL
LIN {X 0,Y 239.689,Z 831.196,A -85,B 0,C 180,E1 18082.267,E2 18082.267} C_VEL
LIN {X 0,Y 230.485,Z 866.361,A -85,B 0,C 180,E1 18090.47,E2 18090.47} C_VEL
LIN {X 0,Y 224.25,Z 888.299,A -85,B 0,C 180,E1 18101.089,E2 18101.089} C_VEL
LIN {X 0,Y 223.437,Z 896.465,A -85,B 0,C 180,E1 18113.511,E2 18113.511} C_VEL
LIN {X 0,Y 229.573,Z 889.984,A -85,B 0,C 180,E1 18125.337,E2 18125.337} C_VEL
LIN {X 0,Y 241.847,Z 869.198,A -85,B 0,C 180,E1 18135.578,E2 18135.578} C_VEL
LIN {X 0,Y 252.879,Z 840.629,A -85,B 0,C 180,E1 18142.633,E2 18142.633} C_VEL
LIN {X 0,Y 247.833,Z 809.077,A -85,B 0,C 180,E1 18150.919,E2 18150.919} C_VEL
LIN {X 0,Y 234.468,Z 780.549,A -85,B 0,C 180,E1 18160.518,E2 18160.518} C_VEL
LIN {X 0,Y 222.235,Z 761.883,A -85,B 0,C 180,E1 18170.662,E2 18170.662} C_VEL
LIN {X 0,Y 219.047,Z 754.81,A -85,B 0,C 180,E1 18178.01,E2 18178.01} C_VEL
LIN {X 0,Y 217.994,Z 756.33,A -85,B 0,C 180,E1 18192.861,E2 18192.861} C_VEL
LIN {X 0,Y 224.376,Z 766.453,A -85,B 0,C 180,E1 18201.317,E2 18201.317} C_VEL
LIN {X 0,Y 238.437,Z 785.956,A -85,B 0,C 180,E1 18211.005,E2 18211.005} C_VEL
LIN {X 0,Y 255.757,Z 819.376,A -85,B 0,C 180,E1 18219.96,E2 18219.96} C_VEL
LIN {X 0,Y 261.704,Z 847.711,A -85,B 0,C 180,E1 18224.98,E2 18224.98} C_VEL
LIN {X 0,Y 246.214,Z 892.772,A -85,B 0,C 180,E1 18230.82,E2 18230.82} C_VEL
LIN {X 0,Y 230.448,Z 929.123,A -85,B 0,C 180,E1 18240.404,E2 18240.404} C_VEL
LIN {X 0,Y 221.768,Z 952.817,A -85,B 0,C 180,E1 18253.078,E2 18253.078} C_VEL
LIN {X 0,Y 221.507,Z 961.422,A -85,B 0,C 180,E1 18264.103,E2 18264.103} C_VEL
LIN {X 0,Y 221.869,Z 960.434,A -85,B 0,C 180,E1 18273.923,E2 18273.923} C_VEL
LIN {X 0,Y 222.169,Z 945.547,A -85,B 0,C 180,E1 18286.765,E2 18286.765} C_VEL
LIN {X 0,Y 228.699,Z 916.452,A -85,B 0,C 180,E1 18298.217,E2 18298.217} C_VEL
LIN {X 0,Y 239.665,Z 875.497,A -85,B 0,C 180,E1 18306.699,E2 18306.699} C_VEL
LIN {X 0,Y 246.85,Z 834.071,A -85,B 0,C 180,E1 18311.348,E2 18311.348} C_VEL
LIN {X 0,Y 230.535,Z 784.913,A -85,B 0,C 180,E1 18316.931,E2 18316.931} C_VEL
LIN {X 0,Y 216.086,Z 754.81,A -85,B 0,C 180,E1 18321.481,E2 18321.481} C_VEL
LIN {X 0,Y 216.824,Z 754.81,A -85,B 0,C 180,E1 18337.365,E2 18337.365} C_VEL
LIN {X 0,Y 218.092,Z 754.81,A -85,B 0,C 180,E1 18349.987,E2 18349.987} C_VEL
LIN {X 0,Y 219.069,Z 754.81,A -85,B 0,C 180,E1 18361.99,E2 18361.99} C_VEL
LIN {X 0,Y 217.284,Z 754.81,A -85,B 0,C 180,E1 18376.91,E2 18376.91} C_VEL
LIN {X 0,Y 216.452,Z 754.81,A -85,B 0,C 180,E1 18385.921,E2 18385.921} C_VEL
LIN {X 0,Y 207.688,Z 754.81,A -85,B 0,C 180,E1 18395.24,E2 18395.24} C_VEL
LIN {X 0,Y 207.683,Z 754.81,A -85,B 0,C 180,E1 18410.115,E2 18410.115} C_VEL
LIN {X 0,Y 208.393,Z 754.81,A -85,B 0,C 180,E1 18425.555,E2 18425.555} C_VEL
LIN {X 0,Y 208.968,Z 756.743,A -85,B 0,C 180,E1 18428.447,E2 18428.447} C_VEL
LIN {X 0,Y 227.515,Z 798.01,A -85,B 0,C 180,E1 18435.295,E2 18435.295} C_VEL
LIN {X 0,Y 232.387,Z 831.432,A -85,B 0,C 180,E1 18441.264,E2 18441.264} C_VEL
LIN {X 0,Y 223.234,Z 866.304,A -85,B 0,C 180,E1 18449.512,E2 18449.512} C_VEL
